LIN {X 0,Y 468.398,Z 466.939,A -85,B 0,C 180,E1 -7680.673,E2 -7680.673} C_VEL
LIN {X 0,Y 468.738,Z 461.358,A -85,B 0,C 180,E1 -7682.899,E2 -7682.899} C_VEL
LIN {X 0,Y 469.168,Z 453.805,A -85,B 0,C 180,E1 -7686.011,E2 -7686.011} C_VEL
LIN {X 0,Y 469.442,Z 448.312,A -85,B 0,C 180,E1 -7688.366,E2 -7688.366} C_VEL
LIN {X 0,Y 469.134,Z 444.309,A -85,B 0,C 180,E1 -7690.18,E2 -7690.18} C_VEL
LIN {X 0,Y 467.968,Z 437.991,A -85,B 0,C 180,E1 -7693.233,E2 -7693.233} C_VEL
LIN {X 0,Y 467.592,Z 435.867,A -85,B 0,C 180,E1 -7694.351,E2 -7694.351} C_VEL
LIN {X 0,Y 467.62,Z 435.861,A -85,B 0,C 180,E1 -7697.443,E2 -7697.443} C_VEL
LIN {X 0,Y 467.578,Z 435.869,A -85,B 0,C 180,E1 -7700.855,E2 -7700.855} C_VEL
LIN {X 0,Y 467.557,Z 435.868,A -85,B 0,C 180,E1 -7704.26,E2 -7704.26} C_VEL
LIN {X 0,Y 467.577,Z 435.869,A -85,B 0,C 180,E1 -7707.32,E2 -7707.32} C_VEL
LIN {X 0,Y 467.573,Z 435.868,A -85,B 0,C 180,E1 -7710.665,E2 -7710.665} C_VEL
LIN {X 0,Y 467.622,Z 435.862,A -85,B 0,C 180,E1 -7713.2,E2 -7713.2} C_VEL
LIN {X 0,Y 467.587,Z 435.866,A -85,B 0,C 180,E1 -7716.468,E2 -7716.468} C_VEL
LIN {X 0,Y 467.617,Z 435.862,A -85,B 0,C 180,E1 -7719.777,E2 -7719.777} C_VEL
LIN {X 0,Y 467.603,Z 435.866,A -85,B 0,C 180,E1 -7722.507,E2 -7722.507} C_VEL
LIN {X 0,Y 467.599,Z 435.866,A -85,B 0,C 180,E1 -7725.196,E2 -7725.196} C_VEL
LIN {X 0,Y 467.65,Z 435.858,A -85,B 0,C 180,E1 -7727.855,E2 -7727.855} C_VEL
LIN {X 0,Y 467.676,Z 435.854,A -85,B 0,C 180,E1 -7731.357,E2 -7731.357} C_VEL
LIN {X 0,Y 467.738,Z 435.847,A -85,B 0,C 180,E1 -7733.963,E2 -7733.963} C_VEL
LIN {X 0,Y 467.854,Z 435.833,A -85,B 0,C 180,E1 -7737.417,E2 -7737.417} C_VEL
LIN {X 0,Y 467.875,Z 435.829,A -85,B 0,C 180,E1 -7740,E2 -7740} C_VEL
LIN {X 0,Y 467.855,Z 435.833,A -85,B 0,C 180,E1 -7742.583,E2 -7742.583} C_VEL
LIN {X 0,Y 467.748,Z 435.848,A -85,B 0,C 180,E1 -7746.038,E2 -7746.038} C_VEL
LIN {X 0,Y 467.676,Z 435.857,A -85,B 0,C 180,E1 -7748.643,E2 -7748.643} C_VEL
LIN {X 0,Y 467.649,Z 435.858,A -85,B 0,C 180,E1 -7752.146,E2 -7752.146} C_VEL
LIN {X 0,Y 467.633,Z 435.861,A -85,B 0,C 180,E1 -7755.695,E2 -7755.695} C_VEL
LIN {X 0,Y 467.612,Z 435.863,A -85,B 0,C 180,E1 -7758.765,E2 -7758.765} C_VEL
LIN {X 0,Y 467.575,Z 435.867,A -85,B 0,C 180,E1 -7761.269,E2 -7761.269} C_VEL
LIN {X 0,Y 467.568,Z 435.871,A -85,B 0,C 180,E1 -7763.944,E2 -7763.944} C_VEL
LIN {X 0,Y 467.612,Z 435.862,A -85,B 0,C 180,E1 -7766.801,E2 -7766.801} C_VEL
LIN {X 0,Y 467.55,Z 435.871,A -85,B 0,C 180,E1 -7769.739,E2 -7769.739} C_VEL
LIN {X 0,Y 467.58,Z 435.867,A -85,B 0,C 180,E1 -7772.759,E2 -7772.759} C_VEL
LIN {X 0,Y 467.553,Z 435.871,A -85,B 0,C 180,E1 -7775.89,E2 -7775.89} C_VEL
LIN {X 0,Y 467.579,Z 435.867,A -85,B 0,C 180,E1 -7779.145,E2 -7779.145} C_VEL
LIN {X 0,Y 467.584,Z 435.867,A -85,B 0,C 180,E1 -7782.568,E2 -7782.568} C_VEL
LIN {X 0,Y 467.569,Z 435.866,A -85,B 0,C 180,E1 -7785.054,E2 -7785.054} C_VEL
LIN {X 0,Y 467.587,Z 435.867,A -85,B 0,C 180,E1 -7787.441,E2 -7787.441} C_VEL
LIN {X 0,Y 467.614,Z 435.862,A -85,B 0,C 180,E1 -7790.859,E2 -7790.859} C_VEL
LIN {X 0,Y 467.563,Z 435.869,A -85,B 0,C 180,E1 -7794.261,E2 -7794.261} C_VEL
LIN {X 0,Y 467.583,Z 435.866,A -85,B 0,C 180,E1 -7797.322,E2 -7797.322} C_VEL
LIN {X 0,Y 467.579,Z 435.867,A -85,B 0,C 180,E1 -7800.666,E2 -7800.666} C_VEL
LIN {X 0,Y 467.618,Z 435.861,A -85,B 0,C 180,E1 -7803.2,E2 -7803.2} C_VEL
LIN {X 0,Y 467.595,Z 435.865,A -85,B 0,C 180,E1 -7806.469,E2 -7806.469} C_VEL
LIN {X 0,Y 467.626,Z 435.862,A -85,B 0,C 180,E1 -7809.778,E2 -7809.778} C_VEL
LIN {X 0,Y 467.61,Z 435.861,A -85,B 0,C 180,E1 -7812.507,E2 -7812.507} C_VEL
LIN {X 0,Y 467.6,Z 435.863,A -85,B 0,C 180,E1 -7815.432,E2 -7815.432} C_VEL
LIN {X 0,Y 466.931,Z 435.948,A -85,B 0,C 180,E1 -7816.152,E2 -7816.152} C_VEL
LIN {X 0,Y 464.087,Z 436.304,A -85,B 0,C 180,E1 -7817.32,E2 -7817.32} C_VEL
LIN {X 0,Y 461.687,Z 436.602,A -85,B 0,C 180,E1 -7818.262,E2 -7818.262} C_VEL
LIN {X 0,Y 460.66,Z 436.73,A -85,B 0,C 180,E1 -7818.99,E2 -7818.99} C_VEL
LIN {X 0,Y 460.578,Z 436.738,A -85,B 0,C 180,E1 -7819.236,E2 -7819.236} C_VEL
LIN {X 0,Y 460.673,Z 436.727,A -85,B 0,C 180,E1 -7822.588,E2 -7822.588} C_VEL
LIN {X 0,Y 460.694,Z 436.724,A -85,B 0,C 180,E1 -7824.748,E2 -7824.748} C_VEL
LIN {X 0,Y 460.828,Z 436.709,A -85,B 0,C 180,E1 -7827.378,E2 -7827.378} C_VEL
LIN {X 0,Y 460.857,Z 436.703,A -85,B 0,C 180,E1 -7830,E2 -7830} C_VEL
LIN {X 0,Y 460.804,Z 436.711,A -85,B 0,C 180,E1 -7832.622,E2 -7832.622} C_VEL
LIN {X 0,Y 460.712,Z 436.722,A -85,B 0,C 180,E1 -7836.13,E2 -7836.13} C_VEL
LIN {X 0,Y 460.625,Z 436.733,A -85,B 0,C 180,E1 -7838.776,E2 -7838.776} C_VEL
LIN {X 0,Y 460.617,Z 436.734,A -85,B 0,C 180,E1 -7842.445,E2 -7842.445} C_VEL
LIN {X 0,Y 460.603,Z 436.736,A -85,B 0,C 180,E1 -7845.997,E2 -7845.997} C_VEL
LIN {X 0,Y 460.574,Z 436.741,A -85,B 0,C 180,E1 -7848.901,E2 -7848.901} C_VEL
LIN {X 0,Y 460.518,Z 436.749,A -85,B 0,C 180,E1 -7851.485,E2 -7851.485} C_VEL
LIN {X 0,Y 460.545,Z 436.743,A -85,B 0,C 180,E1 -7854.332,E2 -7854.332} C_VEL
LIN {X 0,Y 460.581,Z 436.74,A -85,B 0,C 180,E1 -7857.243,E2 -7857.243} C_VEL
LIN {X 0,Y 460.512,Z 436.748,A -85,B 0,C 180,E1 -7860.239,E2 -7860.239} C_VEL
LIN {X 0,Y 460.505,Z 436.748,A -85,B 0,C 180,E1 -7863.326,E2 -7863.326} C_VEL
LIN {X 0,Y 460.311,Z 436.774,A -85,B 0,C 180,E1 -7865.981,E2 -7865.981} C_VEL
LIN {X 0,Y 459.97,Z 436.818,A -85,B 0,C 180,E1 -7868.808,E2 -7868.808} C_VEL
LIN {X 0,Y 459.875,Z 438.549,A -85,B 0,C 180,E1 -7871.081,E2 -7871.081} C_VEL
LIN {X 0,Y 459.846,Z 441.335,A -85,B 0,C 180,E1 -7874.084,E2 -7874.084} C_VEL
LIN {X 0,Y 459.801,Z 444.258,A -85,B 0,C 180,E1 -7877.194,E2 -7877.194} C_VEL
LIN {X 0,Y 459.741,Z 446.977,A -85,B 0,C 180,E1 -7880.055,E2 -7880.055} C_VEL
LIN {X 0,Y 459.739,Z 450.158,A -85,B 0,C 180,E1 -7883.225,E2 -7883.225} C_VEL
LIN {X 0,Y 463.705,Z 464.798,A -85,B 0,C 180,E1 -7883.796,E2 -7883.796} C_VEL
LIN {X 0,Y 464.998,Z 471.275,A -85,B 0,C 180,E1 -7884.091,E2 -7884.091} C_VEL
LIN {X 0,Y 464.463,Z 485.389,A -85,B 0,C 180,E1 -7884.736,E2 -7884.736} C_VEL
LIN {X 0,Y 463.818,Z 498.227,A -85,B 0,C 180,E1 -7885.505,E2 -7885.505} C_VEL
LIN {X 0,Y 463.147,Z 510.816,A -85,B 0,C 180,E1 -7886.457,E2 -7886.457} C_VEL
LIN {X 0,Y 462.369,Z 523.07,A -85,B 0,C 180,E1 -7887.602,E2 -7887.602} C_VEL
LIN {X 0,Y 461.745,Z 533.858,A -85,B 0,C 180,E1 -7888.835,E2 -7888.835} C_VEL
LIN {X 0,Y 461.179,Z 543.327,A -85,B 0,C 180,E1 -7890.144,E2 -7890.144} C_VEL
LIN {X 0,Y 460.683,Z 551.611,A -85,B 0,C 180,E1 -7891.527,E2 -7891.527} C_VEL
LIN {X 0,Y 460.316,Z 558.783,A -85,B 0,C 180,E1 -7892.985,E2 -7892.985} C_VEL
LIN {X 0,Y 460.008,Z 565.432,A -85,B 0,C 180,E1 -7894.673,E2 -7894.673} C_VEL
LIN {X 0,Y 459.828,Z 569.82,A -85,B 0,C 180,E1 -7896.107,E2 -7896.107} C_VEL
LIN {X 0,Y 459.652,Z 573.148,A -85,B 0,C 180,E1 -7897.527,E2 -7897.527} C_VEL
LIN {X 0,Y 459.541,Z 576.153,A -85,B 0,C 180,E1 -7899.405,E2 -7899.405} C_VEL
LIN {X 0,Y 459.512,Z 577.582,A -85,B 0,C 180,E1 -7901.265,E2 -7901.265} C_VEL
LIN {X 0,Y 459.48,Z 577.505,A -85,B 0,C 180,E1 -7903.105,E2 -7903.105} C_VEL
LIN {X 0,Y 459.542,Z 575.992,A -85,B 0,C 180,E1 -7904.93,E2 -7904.93} C_VEL
LIN {X 0,Y 459.658,Z 573.047,A -85,B 0,C 180,E1 -7906.741,E2 -7906.741} C_VEL
LIN {X 0,Y 459.847,Z 570.13,A -85,B 0,C 180,E1 -7907.991,E2 -7907.991} C_VEL
LIN {X 0,Y 460.019,Z 565.795,A -85,B 0,C 180,E1 -7909.436,E2 -7909.436} C_VEL
LIN {X 0,Y 460.316,Z 560.71,A -85,B 0,C 180,E1 -7910.775,E2 -7910.775} C_VEL
LIN {X 0,Y 460.662,Z 553.602,A -85,B 0,C 180,E1 -7912.304,E2 -7912.304} C_VEL
LIN {X 0,Y 461.186,Z 545.878,A -85,B 0,C 180,E1 -7913.657,E2 -7913.657} C_VEL
LIN {X 0,Y 461.679,Z 536.828,A -85,B 0,C 180,E1 -7914.978,E2 -7914.978} C_VEL
LIN {X 0,Y 462.26,Z 527.811,A -85,B 0,C 180,E1 -7916.077,E2 -7916.077} C_VEL
LIN {X 0,Y 462.946,Z 517.097,A -85,B 0,C 180,E1 -7917.172,E2 -7917.172} C_VEL
LIN {X 0,Y 463.623,Z 505.448,A -85,B 0,C 180,E1 -7918.154,E2 -7918.154} C_VEL
LIN {X 0,Y 464.273,Z 493.279,A -85,B 0,C 180,E1 -7918.985,E2 -7918.985} C_VEL
LIN {X 0,Y 464.898,Z 479.944,A -85,B 0,C 180,E1 -7919.701,E2 -7919.701} C_VEL
LIN {X 0,Y 465.049,Z 470.104,A -85,B 0,C 180,E1 -7920.122,E2 -7920.122} C_VEL
LIN {X 0,Y 461.6,Z 457.575,A -85,B 0,C 180,E1 -7920.692,E2 -7920.692} C_VEL
LIN {X 0,Y 459.896,Z 451.959,A -85,B 0,C 180,E1 -7920.93,E2 -7920.93} C_VEL
LIN {X 0,Y 460.184,Z 449.053,A -85,B 0,C 180,E1 -7924.379,E2 -7924.379} C_VEL
LIN {X 0,Y 460.258,Z 446.91,A -85,B 0,C 180,E1 -7927.016,E2 -7927.016} C_VEL
LIN {X 0,Y 460.23,Z 444.85,A -85,B 0,C 180,E1 -7929.67,E2 -7929.67} C_VEL
LIN {X 0,Y 460.37,Z 442.807,A -85,B 0,C 180,E1 -7932.341,E2 -7932.341} C_VEL
LIN {X 0,Y 460.427,Z 440.21,A -85,B 0,C 180,E1 -7935.947,E2 -7935.947} C_VEL
LIN {X 0,Y 460.603,Z 438.172,A -85,B 0,C 180,E1 -7938.916,E2 -7938.916} C_VEL
LIN {X 0,Y 460.5,Z 436.752,A -85,B 0,C 180,E1 -7941.486,E2 -7941.486} C_VEL
LIN {X 0,Y 460.537,Z 436.747,A -85,B 0,C 180,E1 -7944.332,E2 -7944.332} C_VEL
LIN {X 0,Y 460.578,Z 436.74,A -85,B 0,C 180,E1 -7947.243,E2 -7947.243} C_VEL
LIN {X 0,Y 460.522,Z 436.748,A -85,B 0,C 180,E1 -7950.239,E2 -7950.239} C_VEL
LIN {X 0,Y 460.524,Z 436.746,A -85,B 0,C 180,E1 -7953.325,E2 -7953.325} C_VEL
LIN {X 0,Y 460.474,Z 436.753,A -85,B 0,C 180,E1 -7956.53,E2 -7956.53} C_VEL
LIN {X 0,Y 460.572,Z 436.743,A -85,B 0,C 180,E1 -7959.858,E2 -7959.858} C_VEL
LIN {X 0,Y 460.544,Z 436.746,A -85,B 0,C 180,E1 -7962.179,E2 -7962.179} C_VEL
LIN {X 0,Y 460.701,Z 437.663,A -85,B 0,C 180,E1 -7963.352,E2 -7963.352} C_VEL
LIN {X 0,Y 461.163,Z 440.423,A -85,B 0,C 180,E1 -7965.747,E2 -7965.747} C_VEL
LIN {X 0,Y 461.796,Z 443.856,A -85,B 0,C 180,E1 -7968.221,E2 -7968.221} C_VEL
LIN {X 0,Y 462.269,Z 447.226,A -85,B 0,C 180,E1 -7970.318,E2 -7970.318} C_VEL
LIN {X 0,Y 462.362,Z 450.715,A -85,B 0,C 180,E1 -7972.224,E2 -7972.224} C_VEL
LIN {X 0,Y 461.729,Z 457.028,A -85,B 0,C 180,E1 -7975.279,E2 -7975.279} C_VEL
LIN {X 0,Y 461.397,Z 462.642,A -85,B 0,C 180,E1 -7977.784,E2 -7977.784} C_VEL
LIN {X 0,Y 460.967,Z 469.887,A -85,B 0,C 180,E1 -7980.799,E2 -7980.799} C_VEL
LIN {X 0,Y 460.603,Z 478.552,A -85,B 0,C 180,E1 -7984.189,E2 -7984.189} C_VEL
LIN {X 0,Y 460.323,Z 487.611,A -85,B 0,C 180,E1 -7987.562,E2 -7987.562} C_VEL
LIN {X 0,Y 460.101,Z 497.269,A -85,B 0,C 180,E1 -7991.036,E2 -7991.036} C_VEL
LIN {X 0,Y 463.252,Z 515.79,A -85,B 0,C 180,E1 -7991.68,E2 -7991.68} C_VEL
LIN {X 0,Y 464.612,Z 524.172,A -85,B 0,C 180,E1 -7992.049,E2 -7992.049} C_VEL
LIN {X 0,Y 463.983,Z 537.899,A -85,B 0,C 180,E1 -7992.69,E2 -7992.69} C_VEL
LIN {X 0,Y 463.294,Z 550.907,A -85,B 0,C 180,E1 -7993.476,E2 -7993.476} C_VEL
LIN {X 0,Y 462.523,Z 563.982,A -85,B 0,C 180,E1 -7994.466,E2 -7994.466} C_VEL
LIN {X 0,Y 461.782,Z 575.862,A -85,B 0,C 180,E1 -7995.569,E2 -7995.569} C_VEL
LIN {X 0,Y 461.204,Z 586.667,A -85,B 0,C 180,E1 -7996.787,E2 -7996.787} C_VEL
LIN {X 0,Y 460.751,Z 596.45,A -85,B 0,C 180,E1 -7998.117,E2 -7998.117} C_VEL
LIN {X 0,Y 460.226,Z 605.805,A -85,B 0,C 180,E1 -7999.664,E2 -7999.664} C_VEL
LIN {X 0,Y 459.939,Z 613.344,A -85,B 0,C 180,E1 -8001.211,E2 -8001.211} C_VEL
LIN {X 0,Y 459.733,Z 620.127,A -85,B 0,C 180,E1 -8002.975,E2 -8002.975} C_VEL
LIN {X 0,Y 459.694,Z 625.223,A -85,B 0,C 180,E1 -8004.737,E2 -8004.737} C_VEL
LIN {X 0,Y 459.645,Z 628.777,A -85,B 0,C 180,E1 -8006.494,E2 -8006.494} C_VEL
LIN {X 0,Y 459.624,Z 630.897,A -85,B 0,C 180,E1 -8008.248,E2 -8008.248} C_VEL
LIN {X 0,Y 459.528,Z 631.621,A -85,B 0,C 180,E1 -8010,E2 -8010} C_VEL
LIN {X 0,Y 459.624,Z 630.975,A -85,B 0,C 180,E1 -8011.752,E2 -8011.752} C_VEL
LIN {X 0,Y 459.613,Z 628.939,A -85,B 0,C 180,E1 -8013.507,E2 -8013.507} C_VEL
LIN {X 0,Y 459.672,Z 625.476,A -85,B 0,C 180,E1 -8015.263,E2 -8015.263} C_VEL
LIN {X 0,Y 459.731,Z 620.478,A -85,B 0,C 180,E1 -8017.025,E2 -8017.025} C_VEL
LIN {X 0,Y 459.939,Z 613.811,A -85,B 0,C 180,E1 -8018.789,E2 -8018.789} C_VEL
LIN {X 0,Y 460.236,Z 606.382,A -85,B 0,C 180,E1 -8020.336,E2 -8020.336} C_VEL
LIN {X 0,Y 460.746,Z 597.146,A -85,B 0,C 180,E1 -8021.883,E2 -8021.883} C_VEL
LIN {X 0,Y 461.219,Z 587.487,A -85,B 0,C 180,E1 -8023.213,E2 -8023.213} C_VEL
LIN {X 0,Y 461.897,Z 576.811,A -85,B 0,C 180,E1 -8024.427,E2 -8024.427} C_VEL
LIN {X 0,Y 462.614,Z 565.044,A -85,B 0,C 180,E1 -8025.531,E2 -8025.531} C_VEL
LIN {X 0,Y 463.39,Z 552.023,A -85,B 0,C 180,E1 -8026.521,E2 -8026.521} C_VEL
LIN {X 0,Y 464.056,Z 539.426,A -85,B 0,C 180,E1 -8027.283,E2 -8027.283} C_VEL
LIN {X 0,Y 464.621,Z 525.111,A -85,B 0,C 180,E1 -8027.95,E2 -8027.95} C_VEL
LIN {X 0,Y 462.452,Z 511.225,A -85,B 0,C 180,E1 -8028.512,E2 -8028.512} C_VEL
LIN {X 0,Y 460.134,Z 499.005,A -85,B 0,C 180,E1 -8028.892,E2 -8028.892} C_VEL
LIN {X 0,Y 460.377,Z 490.633,A -85,B 0,C 180,E1 -8031.963,E2 -8031.963} C_VEL
LIN {X 0,Y 460.741,Z 481.777,A -85,B 0,C 180,E1 -8035.283,E2 -8035.283} C_VEL
LIN {X 0,Y 461.037,Z 474.214,A -85,B 0,C 180,E1 -8038.2,E2 -8038.2} C_VEL
LIN {X 0,Y 461.541,Z 465.915,A -85,B 0,C 180,E1 -8041.491,E2 -8041.491} C_VEL
LIN {X 0,Y 461.932,Z 457.996,A -85,B 0,C 180,E1 -8044.757,E2 -8044.757} C_VEL
LIN {X 0,Y 462.425,Z 450.94,A -85,B 0,C 180,E1 -8047.786,E2 -8047.786} C_VEL
LIN {X 0,Y 462.324,Z 446.742,A -85,B 0,C 180,E1 -8049.676,E2 -8049.676} C_VEL
LIN {X 0,Y 461.467,Z 441.777,A -85,B 0,C 180,E1 -8052.074,E2 -8052.074} C_VEL
LIN {X 0,Y 460.54,Z 436.746,A -85,B 0,C 180,E1 -8054.657,E2 -8054.657} C_VEL
LIN {X 0,Y 460.543,Z 436.743,A -85,B 0,C 180,E1 -8057.821,E2 -8057.821} C_VEL
LIN {X 0,Y 460.54,Z 436.744,A -85,B 0,C 180,E1 -8061.102,E2 -8061.102} C_VEL
LIN {X 0,Y 460.508,Z 436.748,A -85,B 0,C 180,E1 -8064.554,E2 -8064.554} C_VEL
LIN {X 0,Y 460.528,Z 436.744,A -85,B 0,C 180,E1 -8067.715,E2 -8067.715} C_VEL
LIN {X 0,Y 460.542,Z 436.744,A -85,B 0,C 180,E1 -8070.769,E2 -8070.769} C_VEL
LIN {X 0,Y 460.562,Z 436.741,A -85,B 0,C 180,E1 -8073.735,E2 -8073.735} C_VEL
LIN {X 0,Y 460.54,Z 436.744,A -85,B 0,C 180,E1 -8076.624,E2 -8076.624} C_VEL
LIN {X 0,Y 460.546,Z 436.745,A -85,B 0,C 180,E1 -8079.453,E2 -8079.453} C_VEL
LIN {X 0,Y 460.553,Z 436.741,A -85,B 0,C 180,E1 -8082.23,E2 -8082.23} C_VEL
LIN {X 0,Y 460.558,Z 436.743,A -85,B 0,C 180,E1 -8084.965,E2 -8084.965} C_VEL
LIN {X 0,Y 460.607,Z 436.736,A -85,B 0,C 180,E1 -8088.559,E2 -8088.559} C_VEL
LIN {X 0,Y 460.688,Z 436.726,A -85,B 0,C 180,E1 -8092.109,E2 -8092.109} C_VEL
LIN {X 0,Y 460.692,Z 436.727,A -85,B 0,C 180,E1 -8094.748,E2 -8094.748} C_VEL
LIN {X 0,Y 460.819,Z 436.71,A -85,B 0,C 180,E1 -8097.378,E2 -8097.378} C_VEL
LIN {X 0,Y 460.846,Z 436.704,A -85,B 0,C 180,E1 -8100,E2 -8100} C_VEL
LIN {X 0,Y 460.82,Z 436.71,A -85,B 0,C 180,E1 -8102.623,E2 -8102.623} C_VEL
LIN {X 0,Y 460.712,Z 436.724,A -85,B 0,C 180,E1 -8106.13,E2 -8106.13} C_VEL
LIN {X 0,Y 460.623,Z 436.734,A -85,B 0,C 180,E1 -8108.776,E2 -8108.776} C_VEL
LIN {X 0,Y 460.607,Z 436.737,A -85,B 0,C 180,E1 -8112.445,E2 -8112.445} C_VEL
LIN {X 0,Y 460.594,Z 436.738,A -85,B 0,C 180,E1 -8115.998,E2 -8115.998} C_VEL
LIN {X 0,Y 460.565,Z 436.74,A -85,B 0,C 180,E1 -8118.902,E2 -8118.902} C_VEL
LIN {X 0,Y 460.511,Z 436.747,A -85,B 0,C 180,E1 -8121.486,E2 -8121.486} C_VEL
LIN {X 0,Y 460.538,Z 436.745,A -85,B 0,C 180,E1 -8124.333,E2 -8124.333} C_VEL
LIN {X 0,Y 460.568,Z 436.738,A -85,B 0,C 180,E1 -8127.244,E2 -8127.244} C_VEL
LIN {X 0,Y 460.507,Z 436.749,A -85,B 0,C 180,E1 -8130.241,E2 -8130.241} C_VEL
LIN {X 0,Y 460.526,Z 436.746,A -85,B 0,C 180,E1 -8133.325,E2 -8133.325} C_VEL
LIN {X 0,Y 460.475,Z 436.752,A -85,B 0,C 180,E1 -8136.53,E2 -8136.53} C_VEL
LIN {X 0,Y 460.542,Z 436.744,A -85,B 0,C 180,E1 -8138.898,E2 -8138.898} C_VEL
LIN {X 0,Y 460.521,Z 436.747,A -85,B 0,C 180,E1 -8142.182,E2 -8142.182} C_VEL
LIN {X 0,Y 460.515,Z 436.746,A -85,B 0,C 180,E1 -8145.412,E2 -8145.412} C_VEL
LIN {X 0,Y 460.534,Z 436.746,A -85,B 0,C 180,E1 -8148.398,E2 -8148.398} C_VEL
LIN {X 0,Y 460.543,Z 436.744,A -85,B 0,C 180,E1 -8151.269,E2 -8151.269} C_VEL
LIN {X 0,Y 460.514,Z 436.746,A -85,B 0,C 180,E1 -8154.555,E2 -8154.555} C_VEL
LIN {X 0,Y 460.533,Z 436.746,A -85,B 0,C 180,E1 -8157.716,E2 -8157.716} C_VEL
LIN {X 0,Y 460.548,Z 436.743,A -85,B 0,C 180,E1 -8160.77,E2 -8160.77} C_VEL
LIN {X 0,Y 460.565,Z 436.743,A -85,B 0,C 180,E1 -8163.735,E2 -8163.735} C_VEL
LIN {X 0,Y 460.548,Z 436.742,A -85,B 0,C 180,E1 -8166.625,E2 -8166.625} C_VEL
LIN {X 0,Y 460.554,Z 436.743,A -85,B 0,C 180,E1 -8169.453,E2 -8169.453} C_VEL
LIN {X 0,Y 460.561,Z 436.74,A -85,B 0,C 180,E1 -8172.231,E2 -8172.231} C_VEL
LIN {X 0,Y 460.569,Z 436.741,A -85,B 0,C 180,E1 -8174.965,E2 -8174.965} C_VEL
LIN {X 0,Y 460.614,Z 436.734,A -85,B 0,C 180,E1 -8178.56,E2 -8178.56} C_VEL
LIN {X 0,Y 460.578,Z 436.738,A -85,B 0,C 180,E1 -8179.236,E2 -8179.236} C_VEL
LIN {X 0,Y 459.916,Z 436.824,A -85,B 0,C 180,E1 -8179.966,E2 -8179.966} C_VEL
LIN {X 0,Y 457.075,Z 437.179,A -85,B 0,C 180,E1 -8181.152,E2 -8181.152} C_VEL
LIN {X 0,Y 454.682,Z 437.476,A -85,B 0,C 180,E1 -8182.109,E2 -8182.109} C_VEL
LIN {X 0,Y 453.672,Z 437.6,A -85,B 0,C 180,E1 -8182.848,E2 -8182.848} C_VEL
LIN {X 0,Y 453.599,Z 437.608,A -85,B 0,C 180,E1 -8183.098,E2 -8183.098} C_VEL
LIN {X 0,Y 453.666,Z 437.6,A -85,B 0,C 180,E1 -8184.667,E2 -8184.667} C_VEL
LIN {X 0,Y 453.769,Z 437.588,A -85,B 0,C 180,E1 -8187.337,E2 -8187.337} C_VEL
LIN {X 0,Y 453.827,Z 437.579,A -85,B 0,C 180,E1 -8190,E2 -8190} C_VEL
LIN {X 0,Y 453.748,Z 437.59,A -85,B 0,C 180,E1 -8192.663,E2 -8192.663} C_VEL
LIN {X 0,Y 453.678,Z 437.598,A -85,B 0,C 180,E1 -8196.225,E2 -8196.225} C_VEL
LIN {X 0,Y 453.59,Z 437.609,A -85,B 0,C 180,E1 -8198.913,E2 -8198.913} C_VEL
LIN {X 0,Y 453.567,Z 437.613,A -85,B 0,C 180,E1 -8202.529,E2 -8202.529} C_VEL
LIN {X 0,Y 453.548,Z 437.615,A -85,B 0,C 180,E1 -8206.196,E2 -8206.196} C_VEL
LIN {X 0,Y 453.523,Z 437.62,A -85,B 0,C 180,E1 -8209.04,E2 -8209.04} C_VEL
LIN {X 0,Y 453.479,Z 437.623,A -85,B 0,C 180,E1 -8211.836,E2 -8211.836} C_VEL
LIN {X 0,Y 453.516,Z 437.62,A -85,B 0,C 180,E1 -8214.734,E2 -8214.734} C_VEL
LIN {X 0,Y 453.539,Z 437.614,A -85,B 0,C 180,E1 -8217.96,E2 -8217.96} C_VEL
LIN {X 0,Y 453.464,Z 437.624,A -85,B 0,C 180,E1 -8221.524,E2 -8221.524} C_VEL
LIN {X 0,Y 453.437,Z 437.628,A -85,B 0,C 180,E1 -8223.915,E2 -8223.915} C_VEL
LIN {X 0,Y 453.239,Z 437.655,A -85,B 0,C 180,E1 -8226.261,E2 -8226.261} C_VEL
LIN {X 0,Y 452.827,Z 437.821,A -85,B 0,C 180,E1 -8229.518,E2 -8229.518} C_VEL
LIN {X 0,Y 452.81,Z 441.061,A -85,B 0,C 180,E1 -8233.071,E2 -8233.071} C_VEL
LIN {X 0,Y 452.739,Z 443.499,A -85,B 0,C 180,E1 -8235.689,E2 -8235.689} C_VEL
LIN {X 0,Y 452.698,Z 445.841,A -85,B 0,C 180,E1 -8238.174,E2 -8238.174} C_VEL
LIN {X 0,Y 452.619,Z 449.099,A -85,B 0,C 180,E1 -8241.603,E2 -8241.603} C_VEL
LIN {X 0,Y 452.631,Z 450.374,A -85,B 0,C 180,E1 -8242.912,E2 -8242.912} C_VEL
LIN {X 0,Y 457.129,Z 466.893,A -85,B 0,C 180,E1 -8243.596,E2 -8243.596} C_VEL
LIN {X 0,Y 458.231,Z 471.932,A -85,B 0,C 180,E1 -8243.842,E2 -8243.842} C_VEL
LIN {X 0,Y 457.666,Z 486.107,A -85,B 0,C 180,E1 -8244.506,E2 -8244.506} C_VEL
LIN {X 0,Y 456.96,Z 499.267,A -85,B 0,C 180,E1 -8245.315,E2 -8245.315} C_VEL
LIN {X 0,Y 456.219,Z 512.158,A -85,B 0,C 180,E1 -8246.318,E2 -8246.318} C_VEL
LIN {X 0,Y 455.449,Z 523.903,A -85,B 0,C 180,E1 -8247.444,E2 -8247.444} C_VEL
LIN {X 0,Y 454.864,Z 533.613,A -85,B 0,C 180,E1 -8248.569,E2 -8248.569} C_VEL
LIN {X 0,Y 454.225,Z 543.645,A -85,B 0,C 180,E1 -8249.967,E2 -8249.967} C_VEL
LIN {X 0,Y 453.686,Z 551.566,A -85,B 0,C 180,E1 -8251.3,E2 -8251.3} C_VEL
LIN {X 0,Y 453.319,Z 558.831,A -85,B 0,C 180,E1 -8252.783,E2 -8252.783} C_VEL
LIN {X 0,Y 452.979,Z 564.681,A -85,B 0,C 180,E1 -8254.251,E2 -8254.251} C_VEL
LIN {X 0,Y 452.796,Z 569.335,A -85,B 0,C 180,E1 -8255.712,E2 -8255.712} C_VEL
LIN {X 0,Y 452.613,Z 572.925,A -85,B 0,C 180,E1 -8257.158,E2 -8257.158} C_VEL
LIN {X 0,Y 452.473,Z 576.169,A -85,B 0,C 180,E1 -8259.069,E2 -8259.069} C_VEL
LIN {X 0,Y 452.423,Z 577.852,A -85,B 0,C 180,E1 -8260.96,E2 -8260.96} C_VEL
LIN {X 0,Y 452.396,Z 578.052,A -85,B 0,C 180,E1 -8262.832,E2 -8262.832} C_VEL
LIN {X 0,Y 452.461,Z 576.772,A -85,B 0,C 180,E1 -8264.689,E2 -8264.689} C_VEL
LIN {X 0,Y 452.574,Z 574.036,A -85,B 0,C 180,E1 -8266.53,E2 -8266.53} C_VEL
LIN {X 0,Y 452.774,Z 570.99,A -85,B 0,C 180,E1 -8267.925,E2 -8267.925} C_VEL
LIN {X 0,Y 453.005,Z 565.622,A -85,B 0,C 180,E1 -8269.722,E2 -8269.722} C_VEL
LIN {X 0,Y 453.339,Z 560.458,A -85,B 0,C 180,E1 -8271.081,E2 -8271.081} C_VEL
LIN {X 0,Y 453.772,Z 552.92,A -85,B 0,C 180,E1 -8272.681,E2 -8272.681} C_VEL
LIN {X 0,Y 454.288,Z 545.31,A -85,B 0,C 180,E1 -8274.006,E2 -8274.006} C_VEL
LIN {X 0,Y 454.892,Z 536.025,A -85,B 0,C 180,E1 -8275.347,E2 -8275.347} C_VEL
LIN {X 0,Y 455.604,Z 525.772,A -85,B 0,C 180,E1 -8276.573,E2 -8276.573} C_VEL
LIN {X 0,Y 456.313,Z 514.54,A -85,B 0,C 180,E1 -8277.683,E2 -8277.683} C_VEL
LIN {X 0,Y 457.072,Z 501.895,A -85,B 0,C 180,E1 -8278.7,E2 -8278.7} C_VEL
LIN {X 0,Y 457.75,Z 488.595,A -85,B 0,C 180,E1 -8279.552,E2 -8279.552} C_VEL
LIN {X 0,Y 458.416,Z 474.517,A -85,B 0,C 180,E1 -8280.241,E2 -8280.241} C_VEL
LIN {X 0,Y 458.227,Z 470.76,A -85,B 0,C 180,E1 -8280.405,E2 -8280.405} C_VEL
LIN {X 0,Y 454.439,Z 457.521,A -85,B 0,C 180,E1 -8281.038,E2 -8281.038} C_VEL
LIN {X 0,Y 452.821,Z 452.507,A -85,B 0,C 180,E1 -8281.25,E2 -8281.25} C_VEL
LIN {X 0,Y 453.148,Z 449.854,A -85,B 0,C 180,E1 -8284.447,E2 -8284.447} C_VEL
LIN {X 0,Y 453.214,Z 447.722,A -85,B 0,C 180,E1 -8287.126,E2 -8287.126} C_VEL
LIN {X 0,Y 453.186,Z 445.66,A -85,B 0,C 180,E1 -8289.822,E2 -8289.822} C_VEL
LIN {X 0,Y 453.32,Z 443.64,A -85,B 0,C 180,E1 -8292.536,E2 -8292.536} C_VEL
LIN {X 0,Y 453.412,Z 441.053,A -85,B 0,C 180,E1 -8296.201,E2 -8296.201} C_VEL
LIN {X 0,Y 453.593,Z 439.161,A -85,B 0,C 180,E1 -8299.07,E2 -8299.07} C_VEL
LIN {X 0,Y 453.465,Z 437.628,A -85,B 0,C 180,E1 -8301.837,E2 -8301.837} C_VEL
LIN {X 0,Y 453.508,Z 437.621,A -85,B 0,C 180,E1 -8304.735,E2 -8304.735} C_VEL
LIN {X 0,Y 453.533,Z 437.619,A -85,B 0,C 180,E1 -8307.962,E2 -8307.962} C_VEL
LIN {X 0,Y 453.478,Z 437.624,A -85,B 0,C 180,E1 -8310.759,E2 -8310.759} C_VEL
LIN {X 0,Y 453.473,Z 437.625,A -85,B 0,C 180,E1 -8313.913,E2 -8313.913} C_VEL
LIN {X 0,Y 453.466,Z 437.626,A -85,B 0,C 180,E1 -8317.188,E2 -8317.188} C_VEL
LIN {X 0,Y 453.527,Z 437.619,A -85,B 0,C 180,E1 -8319.446,E2 -8319.446} C_VEL
LIN {X 0,Y 453.54,Z 437.897,A -85,B 0,C 180,E1 -8321.945,E2 -8321.945} C_VEL
LIN {X 0,Y 454.016,Z 440.58,A -85,B 0,C 180,E1 -8324.598,E2 -8324.598} C_VEL
LIN {X 0,Y 454.743,Z 444.815,A -85,B 0,C 180,E1 -8327.888,E2 -8327.888} C_VEL
LIN {X 0,Y 455.213,Z 447.406,A -85,B 0,C 180,E1 -8329.577,E2 -8329.577} C_VEL
LIN {X 0,Y 455.415,Z 450.379,A -85,B 0,C 180,E1 -8331.319,E2 -8331.319} C_VEL
LIN {X 0,Y 455.088,Z 454.38,A -85,B 0,C 180,E1 -8333.422,E2 -8333.422} C_VEL
LIN {X 0,Y 454.527,Z 461.11,A -85,B 0,C 180,E1 -8336.612,E2 -8336.612} C_VEL
LIN {X 0,Y 454.112,Z 467.219,A -85,B 0,C 180,E1 -8339.289,E2 -8339.289} C_VEL
LIN {X 0,Y 453.747,Z 474.573,A -85,B 0,C 180,E1 -8342.312,E2 -8342.312} C_VEL
LIN {X 0,Y 453.429,Z 482.105,A -85,B 0,C 180,E1 -8345.261,E2 -8345.261} C_VEL
LIN {X 0,Y 453.169,Z 490.763,A -85,B 0,C 180,E1 -8348.515,E2 -8348.515} C_VEL
LIN {X 0,Y 453.024,Z 496.747,A -85,B 0,C 180,E1 -8350.702,E2 -8350.702} C_VEL
LIN {X 0,Y 456.101,Z 514.227,A -85,B 0,C 180,E1 -8351.338,E2 -8351.338} C_VEL
LIN {X 0,Y 457.77,Z 525.816,A -85,B 0,C 180,E1 -8351.86,E2 -8351.86} C_VEL
LIN {X 0,Y 457.098,Z 538.869,A -85,B 0,C 180,E1 -8352.501,E2 -8352.501} C_VEL
LIN {X 0,Y 456.358,Z 552.055,A -85,B 0,C 180,E1 -8353.332,E2 -8353.332} C_VEL
LIN {X 0,Y 455.539,Z 564.834,A -85,B 0,C 180,E1 -8354.337,E2 -8354.337} C_VEL
LIN {X 0,Y 454.766,Z 576.461,A -85,B 0,C 180,E1 -8355.456,E2 -8355.456} C_VEL
LIN {X 0,Y 454.22,Z 586.157,A -85,B 0,C 180,E1 -8356.58,E2 -8356.58} C_VEL
LIN {X 0,Y 453.755,Z 595.936,A -85,B 0,C 180,E1 -8357.931,E2 -8357.931} C_VEL
LIN {X 0,Y 453.191,Z 605.313,A -85,B 0,C 180,E1 -8359.501,E2 -8359.501} C_VEL
LIN {X 0,Y 452.891,Z 612.871,A -85,B 0,C 180,E1 -8361.073,E2 -8361.073} C_VEL
LIN {X 0,Y 452.651,Z 619.671,A -85,B 0,C 180,E1 -8362.865,E2 -8362.865} C_VEL
LIN {X 0,Y 452.6,Z 624.782,A -85,B 0,C 180,E1 -8364.654,E2 -8364.654} C_VEL
LIN {X 0,Y 452.542,Z 628.348,A -85,B 0,C 180,E1 -8366.439,E2 -8366.439} C_VEL
LIN {X 0,Y 452.532,Z 630.478,A -85,B 0,C 180,E1 -8368.22,E2 -8368.22} C_VEL
LIN {X 0,Y 452.462,Z 631.206,A -85,B 0,C 180,E1 -8370,E2 -8370} C_VEL
LIN {X 0,Y 452.532,Z 630.559,A -85,B 0,C 180,E1 -8371.78,E2 -8371.78} C_VEL
LIN {X 0,Y 452.513,Z 628.519,A -85,B 0,C 180,E1 -8373.562,E2 -8373.562} C_VEL
LIN {X 0,Y 452.583,Z 625.049,A -85,B 0,C 180,E1 -8375.346,E2 -8375.346} C_VEL
LIN {X 0,Y 452.651,Z 620.04,A -85,B 0,C 180,E1 -8377.135,E2 -8377.135} C_VEL
LIN {X 0,Y 452.885,Z 613.358,A -85,B 0,C 180,E1 -8378.927,E2 -8378.927} C_VEL
LIN {X 0,Y 453.207,Z 605.913,A -85,B 0,C 180,E1 -8380.498,E2 -8380.498} C_VEL
LIN {X 0,Y 453.754,Z 596.653,A -85,B 0,C 180,E1 -8382.069,E2 -8382.069} C_VEL
LIN {X 0,Y 454.234,Z 586.972,A -85,B 0,C 180,E1 -8383.419,E2 -8383.419} C_VEL
LIN {X 0,Y 454.912,Z 576.271,A -85,B 0,C 180,E1 -8384.654,E2 -8384.654} C_VEL
LIN {X 0,Y 455.693,Z 564.485,A -85,B 0,C 180,E1 -8385.773,E2 -8385.773} C_VEL
LIN {X 0,Y 456.537,Z 551.444,A -85,B 0,C 180,E1 -8386.776,E2 -8386.776} C_VEL
LIN {X 0,Y 457.214,Z 538.815,A -85,B 0,C 180,E1 -8387.55,E2 -8387.55} C_VEL
LIN {X 0,Y 457.744,Z 524.756,A -85,B 0,C 180,E1 -8388.216,E2 -8388.216} C_VEL
LIN {X 0,Y 455.286,Z 510.21,A -85,B 0,C 180,E1 -8388.819,E2 -8388.819} C_VEL
LIN {X 0,Y 453.084,Z 498.662,A -85,B 0,C 180,E1 -8389.187,E2 -8389.187} C_VEL
LIN {X 0,Y 453.353,Z 490.291,A -85,B 0,C 180,E1 -8392.321,E2 -8392.321} C_VEL
LIN {X 0,Y 453.743,Z 481.472,A -85,B 0,C 180,E1 -8395.701,E2 -8395.701} C_VEL
LIN {X 0,Y 454.136,Z 472.678,A -85,B 0,C 180,E1 -8399.174,E2 -8399.174} C_VEL
LIN {X 0,Y 454.585,Z 465.17,A -85,B 0,C 180,E1 -8402.233,E2 -8402.233} C_VEL
LIN {X 0,Y 455.056,Z 457.584,A -85,B 0,C 180,E1 -8405.44,E2 -8405.44} C_VEL
LIN {X 0,Y 455.461,Z 451.468,A -85,B 0,C 180,E1 -8408.113,E2 -8408.113} C_VEL
LIN {X 0,Y 455.372,Z 448.47,A -85,B 0,C 180,E1 -8409.495,E2 -8409.495} C_VEL
LIN {X 0,Y 454.529,Z 443.161,A -85,B 0,C 180,E1 -8412.082,E2 -8412.082} C_VEL
LIN {X 0,Y 453.507,Z 437.622,A -85,B 0,C 180,E1 -8414.979,E2 -8414.979} C_VEL
LIN {X 0,Y 453.489,Z 437.621,A -85,B 0,C 180,E1 -8418.21,E2 -8418.21} C_VEL
LIN {X 0,Y 453.511,Z 437.621,A -85,B 0,C 180,E1 -8420.79,E2 -8420.79} C_VEL
LIN {X 0,Y 453.451,Z 437.625,A -85,B 0,C 180,E1 -8423.917,E2 -8423.917} C_VEL
LIN {X 0,Y 453.478,Z 437.625,A -85,B 0,C 180,E1 -8427.151,E2 -8427.151} C_VEL
LIN {X 0,Y 453.509,Z 437.62,A -85,B 0,C 180,E1 -8430.271,E2 -8430.271} C_VEL
LIN {X 0,Y 453.508,Z 437.62,A -85,B 0,C 180,E1 -8433.294,E2 -8433.294} C_VEL
LIN {X 0,Y 453.497,Z 437.62,A -85,B 0,C 180,E1 -8436.239,E2 -8436.239} C_VEL
LIN {X 0,Y 453.477,Z 437.624,A -85,B 0,C 180,E1 -8439.117,E2 -8439.117} C_VEL
LIN {X 0,Y 453.505,Z 437.618,A -85,B 0,C 180,E1 -8441.944,E2 -8441.944} C_VEL
LIN {X 0,Y 453.533,Z 437.617,A -85,B 0,C 180,E1 -8444.726,E2 -8444.726} C_VEL
LIN {X 0,Y 453.555,Z 437.615,A -85,B 0,C 180,E1 -8448.379,E2 -8448.379} C_VEL
LIN {X 0,Y 453.645,Z 437.602,A -85,B 0,C 180,E1 -8451.985,E2 -8451.985} C_VEL
LIN {X 0,Y 453.666,Z 437.602,A -85,B 0,C 180,E1 -8454.667,E2 -8454.667} C_VEL
LIN {X 0,Y 453.76,Z 437.589,A -85,B 0,C 180,E1 -8457.337,E2 -8457.337} C_VEL
LIN {X 0,Y 453.816,Z 437.58,A -85,B 0,C 180,E1 -8460,E2 -8460} C_VEL
LIN {X 0,Y 453.761,Z 437.589,A -85,B 0,C 180,E1 -8462.663,E2 -8462.663} C_VEL
LIN {X 0,Y 453.678,Z 437.6,A -85,B 0,C 180,E1 -8466.225,E2 -8466.225} C_VEL
LIN {X 0,Y 453.587,Z 437.61,A -85,B 0,C 180,E1 -8468.914,E2 -8468.914} C_VEL
LIN {X 0,Y 453.557,Z 437.616,A -85,B 0,C 180,E1 -8472.529,E2 -8472.529} C_VEL
LIN {X 0,Y 453.539,Z 437.616,A -85,B 0,C 180,E1 -8476.196,E2 -8476.196} C_VEL
LIN {X 0,Y 453.515,Z 437.619,A -85,B 0,C 180,E1 -8479.041,E2 -8479.041} C_VEL
LIN {X 0,Y 453.472,Z 437.624,A -85,B 0,C 180,E1 -8481.837,E2 -8481.837} C_VEL
LIN {X 0,Y 453.509,Z 437.621,A -85,B 0,C 180,E1 -8484.735,E2 -8484.735} C_VEL
LIN {X 0,Y 453.527,Z 437.62,A -85,B 0,C 180,E1 -8487.96,E2 -8487.96} C_VEL
LIN {X 0,Y 453.463,Z 437.624,A -85,B 0,C 180,E1 -8491.526,E2 -8491.526} C_VEL
LIN {X 0,Y 453.485,Z 437.623,A -85,B 0,C 180,E1 -8494.778,E2 -8494.778} C_VEL
LIN {X 0,Y 453.47,Z 437.625,A -85,B 0,C 180,E1 -8498.311,E2 -8498.311} C_VEL
LIN {X 0,Y 453.492,Z 437.621,A -85,B 0,C 180,E1 -8500.61,E2 -8500.61} C_VEL
LIN {X 0,Y 453.461,Z 437.626,A -85,B 0,C 180,E1 -8503.246,E2 -8503.246} C_VEL
LIN {X 0,Y 453.464,Z 437.628,A -85,B 0,C 180,E1 -8505.78,E2 -8505.78} C_VEL
LIN {X 0,Y 453.515,Z 437.618,A -85,B 0,C 180,E1 -8509.406,E2 -8509.406} C_VEL
LIN {X 0,Y 453.476,Z 437.625,A -85,B 0,C 180,E1 -8512.223,E2 -8512.223} C_VEL
LIN {X 0,Y 453.49,Z 437.622,A -85,B 0,C 180,E1 -8515.223,E2 -8515.223} C_VEL
LIN {X 0,Y 453.469,Z 437.623,A -85,B 0,C 180,E1 -8518.475,E2 -8518.475} C_VEL
LIN {X 0,Y 453.517,Z 437.619,A -85,B 0,C 180,E1 -8521.289,E2 -8521.289} C_VEL
LIN {X 0,Y 453.526,Z 437.617,A -85,B 0,C 180,E1 -8524.285,E2 -8524.285} C_VEL
LIN {X 0,Y 453.482,Z 437.622,A -85,B 0,C 180,E1 -8527.205,E2 -8527.205} C_VEL
LIN {X 0,Y 453.508,Z 437.621,A -85,B 0,C 180,E1 -8530.067,E2 -8530.067} C_VEL
LIN {X 0,Y 453.509,Z 437.618,A -85,B 0,C 180,E1 -8532.876,E2 -8532.876} C_VEL
LIN {X 0,Y 453.517,Z 437.62,A -85,B 0,C 180,E1 -8535.644,E2 -8535.644} C_VEL
LIN {X 0,Y 453.563,Z 437.613,A -85,B 0,C 180,E1 -8538.379,E2 -8538.379} C_VEL
LIN {X 0,Y 453.595,Z 437.609,A -85,B 0,C 180,E1 -8541.087,E2 -8541.087} C_VEL
LIN {X 0,Y 453.599,Z 437.608,A -85,B 0,C 180,E1 -8543.098,E2 -8543.098} C_VEL
LIN {X 0,Y 452.929,Z 437.693,A -85,B 0,C 180,E1 -8543.839,E2 -8543.839} C_VEL
LIN {X 0,Y 449.997,Z 438.057,A -85,B 0,C 180,E1 -8545.041,E2 -8545.041} C_VEL
LIN {X 0,Y 447.581,Z 438.357,A -85,B 0,C 180,E1 -8546.011,E2 -8546.011} C_VEL
LIN {X 0,Y 446.648,Z 438.474,A -85,B 0,C 180,E1 -8546.762,E2 -8546.762} C_VEL
LIN {X 0,Y 446.629,Z 438.476,A -85,B 0,C 180,E1 -8547.015,E2 -8547.015} C_VEL
LIN {X 0,Y 446.797,Z 438.454,A -85,B 0,C 180,E1 -8550,E2 -8550} C_VEL
LIN {X 0,Y 446.695,Z 438.469,A -85,B 0,C 180,E1 -8552.705,E2 -8552.705} C_VEL
LIN {X 0,Y 446.646,Z 438.474,A -85,B 0,C 180,E1 -8556.324,E2 -8556.324} C_VEL
LIN {X 0,Y 446.538,Z 438.489,A -85,B 0,C 180,E1 -8559.055,E2 -8559.055} C_VEL
LIN {X 0,Y 446.525,Z 438.489,A -85,B 0,C 180,E1 -8562.729,E2 -8562.729} C_VEL
LIN {X 0,Y 446.499,Z 438.492,A -85,B 0,C 180,E1 -8566.227,E2 -8566.227} C_VEL
LIN {X 0,Y 446.472,Z 438.497,A -85,B 0,C 180,E1 -8569.303,E2 -8569.303} C_VEL
LIN {X 0,Y 446.421,Z 438.501,A -85,B 0,C 180,E1 -8572.199,E2 -8572.199} C_VEL
LIN {X 0,Y 446.46,Z 438.498,A -85,B 0,C 180,E1 -8575.152,E2 -8575.152} C_VEL
LIN {X 0,Y 446.486,Z 438.493,A -85,B 0,C 180,E1 -8578.178,E2 -8578.178} C_VEL
LIN {X 0,Y 446.415,Z 438.504,A -85,B 0,C 180,E1 -8581.3,E2 -8581.3} C_VEL
LIN {X 0,Y 446.423,Z 438.503,A -85,B 0,C 180,E1 -8583.449,E2 -8583.449} C_VEL
LIN {X 0,Y 446.246,Z 438.526,A -85,B 0,C 180,E1 -8585.641,E2 -8585.641} C_VEL
LIN {X 0,Y 445.84,Z 438.579,A -85,B 0,C 180,E1 -8589.089,E2 -8589.089} C_VEL
LIN {X 0,Y 445.779,Z 439.198,A -85,B 0,C 180,E1 -8590.269,E2 -8590.269} C_VEL
LIN {X 0,Y 445.702,Z 442.144,A -85,B 0,C 180,E1 -8593.502,E2 -8593.502} C_VEL
LIN {X 0,Y 445.652,Z 444.915,A -85,B 0,C 180,E1 -8596.503,E2 -8596.503} C_VEL
LIN {X 0,Y 445.561,Z 447.934,A -85,B 0,C 180,E1 -8599.706,E2 -8599.706} C_VEL
LIN {X 0,Y 445.58,Z 450.827,A -85,B 0,C 180,E1 -8602.639,E2 -8602.639} C_VEL
LIN {X 0,Y 449.724,Z 465.796,A -85,B 0,C 180,E1 -8603.25,E2 -8603.25} C_VEL
LIN {X 0,Y 451.336,Z 472.357,A -85,B 0,C 180,E1 -8603.574,E2 -8603.574} C_VEL
LIN {X 0,Y 450.895,Z 486.252,A -85,B 0,C 180,E1 -8604.24,E2 -8604.24} C_VEL
LIN {X 0,Y 450.207,Z 498.498,A -85,B 0,C 180,E1 -8604.992,E2 -8604.992} C_VEL
LIN {X 0,Y 449.465,Z 511.123,A -85,B 0,C 180,E1 -8605.967,E2 -8605.967} C_VEL
LIN {X 0,Y 448.706,Z 522.319,A -85,B 0,C 180,E1 -8607.024,E2 -8607.024} C_VEL
LIN {X 0,Y 447.965,Z 533.359,A -85,B 0,C 180,E1 -8608.293,E2 -8608.293} C_VEL
LIN {X 0,Y 447.366,Z 542.672,A -85,B 0,C 180,E1 -8609.586,E2 -8609.586} C_VEL
LIN {X 0,Y 446.699,Z 551.659,A -85,B 0,C 180,E1 -8611.092,E2 -8611.092} C_VEL
LIN {X 0,Y 446.316,Z 558.878,A -85,B 0,C 180,E1 -8612.574,E2 -8612.574} C_VEL
LIN {X 0,Y 445.916,Z 565.867,A -85,B 0,C 180,E1 -8614.363,E2 -8614.363} C_VEL
LIN {X 0,Y 445.659,Z 571.17,A -85,B 0,C 180,E1 -8616.154,E2 -8616.154} C_VEL
LIN {X 0,Y 445.486,Z 574.641,A -85,B 0,C 180,E1 -8617.751,E2 -8617.751} C_VEL
LIN {X 0,Y 445.442,Z 576.185,A -85,B 0,C 180,E1 -8618.722,E2 -8618.722} C_VEL
LIN {X 0,Y 445.338,Z 578.095,A -85,B 0,C 180,E1 -8620.646,E2 -8620.646} C_VEL
LIN {X 0,Y 445.352,Z 578.486,A -85,B 0,C 180,E1 -8621.602,E2 -8621.602} C_VEL
LIN {X 0,Y 445.33,Z 578.176,A -85,B 0,C 180,E1 -8623.497,E2 -8623.497} C_VEL
LIN {X 0,Y 445.415,Z 576.428,A -85,B 0,C 180,E1 -8625.377,E2 -8625.377} C_VEL
LIN {X 0,Y 445.608,Z 573.221,A -85,B 0,C 180,E1 -8627.244,E2 -8627.244} C_VEL
LIN {X 0,Y 445.866,Z 568.462,A -85,B 0,C 180,E1 -8629.097,E2 -8629.097} C_VEL
LIN {X 0,Y 446.122,Z 563.863,A -85,B 0,C 180,E1 -8630.479,E2 -8630.479} C_VEL
LIN {X 0,Y 446.439,Z 558.208,A -85,B 0,C 180,E1 -8631.855,E2 -8631.855} C_VEL
LIN {X 0,Y 447.08,Z 550.145,A -85,B 0,C 180,E1 -8633.456,E2 -8633.456} C_VEL
LIN {X 0,Y 447.603,Z 541.769,A -85,B 0,C 180,E1 -8634.82,E2 -8634.82} C_VEL
LIN {X 0,Y 448.314,Z 531.637,A -85,B 0,C 180,E1 -8636.18,E2 -8636.18} C_VEL
LIN {X 0,Y 449.14,Z 520.357,A -85,B 0,C 180,E1 -8637.421,E2 -8637.421} C_VEL
LIN {X 0,Y 449.935,Z 508.267,A -85,B 0,C 180,E1 -8638.514,E2 -8638.514} C_VEL
LIN {X 0,Y 450.714,Z 495.579,A -85,B 0,C 180,E1 -8639.438,E2 -8639.438} C_VEL
LIN {X 0,Y 451.422,Z 482.752,A -85,B 0,C 180,E1 -8640.176,E2 -8640.176} C_VEL
LIN {X 0,Y 451.677,Z 472.836,A -85,B 0,C 180,E1 -8640.633,E2 -8640.633} C_VEL
LIN {X 0,Y 447.973,Z 459.844,A -85,B 0,C 180,E1 -8641.291,E2 -8641.291} C_VEL
LIN {X 0,Y 445.777,Z 453.056,A -85,B 0,C 180,E1 -8641.589,E2 -8641.589} C_VEL
LIN {X 0,Y 446.114,Z 450.646,A -85,B 0,C 180,E1 -8644.518,E2 -8644.518} C_VEL
LIN {X 0,Y 446.173,Z 448.524,A -85,B 0,C 180,E1 -8647.239,E2 -8647.239} C_VEL
LIN {X 0,Y 446.149,Z 446.483,A -85,B 0,C 180,E1 -8649.978,E2 -8649.978} C_VEL
LIN {X 0,Y 446.288,Z 444.463,A -85,B 0,C 180,E1 -8652.736,E2 -8652.736} C_VEL
LIN {X 0,Y 446.406,Z 442.107,A -85,B 0,C 180,E1 -8656.191,E2 -8656.191} C_VEL
LIN {X 0,Y 446.553,Z 440.144,A -85,B 0,C 180,E1 -8659.299,E2 -8659.299} C_VEL
LIN {X 0,Y 446.41,Z 438.53,A -85,B 0,C 180,E1 -8662.2,E2 -8662.2} C_VEL
LIN {X 0,Y 446.452,Z 438.5,A -85,B 0,C 180,E1 -8665.152,E2 -8665.152} C_VEL
LIN {X 0,Y 446.479,Z 438.497,A -85,B 0,C 180,E1 -8668.179,E2 -8668.179} C_VEL
LIN {X 0,Y 446.415,Z 438.504,A -85,B 0,C 180,E1 -8671.3,E2 -8671.3} C_VEL
LIN {X 0,Y 446.426,Z 438.503,A -85,B 0,C 180,E1 -8674.523,E2 -8674.523} C_VEL
LIN {X 0,Y 446.432,Z 438.503,A -85,B 0,C 180,E1 -8678.083,E2 -8678.083} C_VEL
LIN {X 0,Y 446.48,Z 438.644,A -85,B 0,C 180,E1 -8680.927,E2 -8680.927} C_VEL
LIN {X 0,Y 446.955,Z 441.213,A -85,B 0,C 180,E1 -8683.778,E2 -8683.778} C_VEL
LIN {X 0,Y 447.561,Z 444.943,A -85,B 0,C 180,E1 -8686.917,E2 -8686.917} C_VEL
LIN {X 0,Y 448.077,Z 447.696,A -85,B 0,C 180,E1 -8688.84,E2 -8688.84} C_VEL
LIN {X 0,Y 448.435,Z 451.48,A -85,B 0,C 180,E1 -8691.18,E2 -8691.18} C_VEL
LIN {X 0,Y 448.201,Z 455.048,A -85,B 0,C 180,E1 -8693.102,E2 -8693.102} C_VEL
LIN {X 0,Y 447.506,Z 462.369,A -85,B 0,C 180,E1 -8696.656,E2 -8696.656} C_VEL
LIN {X 0,Y 447.063,Z 469.523,A -85,B 0,C 180,E1 -8699.839,E2 -8699.839} C_VEL
LIN {X 0,Y 446.636,Z 476.753,A -85,B 0,C 180,E1 -8702.85,E2 -8702.85} C_VEL
LIN {X 0,Y 446.285,Z 484.652,A -85,B 0,C 180,E1 -8705.976,E2 -8705.976} C_VEL
LIN {X 0,Y 446.056,Z 491.942,A -85,B 0,C 180,E1 -8708.754,E2 -8708.754} C_VEL
LIN {X 0,Y 445.947,Z 496.271,A -85,B 0,C 180,E1 -8710.37,E2 -8710.37} C_VEL
LIN {X 0,Y 448.897,Z 512.219,A -85,B 0,C 180,E1 -8710.951,E2 -8710.951} C_VEL
LIN {X 0,Y 450.925,Z 527.34,A -85,B 0,C 180,E1 -8711.657,E2 -8711.657} C_VEL
LIN {X 0,Y 450.174,Z 541.044,A -85,B 0,C 180,E1 -8712.377,E2 -8712.377} C_VEL
LIN {X 0,Y 449.328,Z 554.759,A -85,B 0,C 180,E1 -8713.298,E2 -8713.298} C_VEL
LIN {X 0,Y 448.482,Z 566.924,A -85,B 0,C 180,E1 -8714.317,E2 -8714.317} C_VEL
LIN {X 0,Y 447.721,Z 578.089,A -85,B 0,C 180,E1 -8715.454,E2 -8715.454} C_VEL
LIN {X 0,Y 447.051,Z 589.162,A -85,B 0,C 180,E1 -8716.824,E2 -8716.824} C_VEL
LIN {X 0,Y 446.509,Z 598.338,A -85,B 0,C 180,E1 -8718.193,E2 -8718.193} C_VEL
LIN {X 0,Y 446.045,Z 607.151,A -85,B 0,C 180,E1 -8719.79,E2 -8719.79} C_VEL
LIN {X 0,Y 445.742,Z 614.278,A -85,B 0,C 180,E1 -8721.386,E2 -8721.386} C_VEL
LIN {X 0,Y 445.575,Z 619.219,A -85,B 0,C 180,E1 -8722.751,E2 -8722.751} C_VEL
LIN {X 0,Y 445.513,Z 622.676,A -85,B 0,C 180,E1 -8723.904,E2 -8723.904} C_VEL
LIN {X 0,Y 445.413,Z 626.314,A -85,B 0,C 180,E1 -8725.475,E2 -8725.475} C_VEL
LIN {X 0,Y 445.454,Z 629.167,A -85,B 0,C 180,E1 -8727.287,E2 -8727.287} C_VEL
LIN {X 0,Y 445.424,Z 630.599,A -85,B 0,C 180,E1 -8729.096,E2 -8729.096} C_VEL
LIN {X 0,Y 445.424,Z 630.639,A -85,B 0,C 180,E1 -8730.904,E2 -8730.904} C_VEL
LIN {X 0,Y 445.451,Z 629.295,A -85,B 0,C 180,E1 -8732.713,E2 -8732.713} C_VEL
LIN {X 0,Y 445.408,Z 626.54,A -85,B 0,C 180,E1 -8734.525,E2 -8734.525} C_VEL
LIN {X 0,Y 445.488,Z 623.065,A -85,B 0,C 180,E1 -8736.067,E2 -8736.067} C_VEL
LIN {X 0,Y 445.58,Z 618.107,A -85,B 0,C 180,E1 -8737.705,E2 -8737.705} C_VEL
LIN {X 0,Y 445.807,Z 612.903,A -85,B 0,C 180,E1 -8739.07,E2 -8739.07} C_VEL
LIN {X 0,Y 446.176,Z 605.442,A -85,B 0,C 180,E1 -8740.666,E2 -8740.666} C_VEL
LIN {X 0,Y 446.641,Z 597.627,A -85,B 0,C 180,E1 -8742.034,E2 -8742.034} C_VEL
LIN {X 0,Y 447.16,Z 588.416,A -85,B 0,C 180,E1 -8743.381,E2 -8743.381} C_VEL
LIN {X 0,Y 447.879,Z 577.888,A -85,B 0,C 180,E1 -8744.657,E2 -8744.657} C_VEL
LIN {X 0,Y 448.654,Z 566.508,A -85,B 0,C 180,E1 -8745.793,E2 -8745.793} C_VEL
LIN {X 0,Y 449.464,Z 553.996,A -85,B 0,C 180,E1 -8746.814,E2 -8746.814} C_VEL
LIN {X 0,Y 450.282,Z 540.915,A -85,B 0,C 180,E1 -8747.666,E2 -8747.666} C_VEL
LIN {X 0,Y 450.928,Z 527.662,A -85,B 0,C 180,E1 -8748.34,E2 -8748.34} C_VEL
LIN {X 0,Y 450.153,Z 521.318,A -85,B 0,C 180,E1 -8748.642,E2 -8748.642} C_VEL
LIN {X 0,Y 447.699,Z 506.913,A -85,B 0,C 180,E1 -8749.216,E2 -8749.216} C_VEL
LIN {X 0,Y 446.021,Z 498.294,A -85,B 0,C 180,E1 -8749.502,E2 -8749.502} C_VEL
LIN {X 0,Y 446.331,Z 489.955,A -85,B 0,C 180,E1 -8752.692,E2 -8752.692} C_VEL
LIN {X 0,Y 446.759,Z 480.798,A -85,B 0,C 180,E1 -8756.276,E2 -8756.276} C_VEL
LIN {X 0,Y 447.186,Z 472.39,A -85,B 0,C 180,E1 -8759.673,E2 -8759.673} C_VEL
LIN {X 0,Y 447.665,Z 464.892,A -85,B 0,C 180,E1 -8762.794,E2 -8762.794} C_VEL
LIN {X 0,Y 448.156,Z 457.423,A -85,B 0,C 180,E1 -8766.02,E2 -8766.02} C_VEL
LIN {X 0,Y 448.494,Z 452.088,A -85,B 0,C 180,E1 -8768.417,E2 -8768.417} C_VEL
LIN {X 0,Y 448.124,Z 447.577,A -85,B 0,C 180,E1 -8770.559,E2 -8770.559} C_VEL
LIN {X 0,Y 446.943,Z 441.272,A -85,B 0,C 180,E1 -8773.778,E2 -8773.778} C_VEL
LIN {X 0,Y 446.464,Z 438.499,A -85,B 0,C 180,E1 -8775.267,E2 -8775.267} C_VEL
LIN {X 0,Y 446.433,Z 438.5,A -85,B 0,C 180,E1 -8778.61,E2 -8778.61} C_VEL
LIN {X 0,Y 446.455,Z 438.499,A -85,B 0,C 180,E1 -8780.974,E2 -8780.974} C_VEL
LIN {X 0,Y 446.416,Z 438.502,A -85,B 0,C 180,E1 -8784.374,E2 -8784.374} C_VEL
LIN {X 0,Y 446.425,Z 438.501,A -85,B 0,C 180,E1 -8787.639,E2 -8787.639} C_VEL
LIN {X 0,Y 446.464,Z 438.498,A -85,B 0,C 180,E1 -8790.792,E2 -8790.792} C_VEL
LIN {X 0,Y 446.472,Z 438.495,A -85,B 0,C 180,E1 -8793.848,E2 -8793.848} C_VEL
LIN {X 0,Y 446.424,Z 438.504,A -85,B 0,C 180,E1 -8796.823,E2 -8796.823} C_VEL
LIN {X 0,Y 446.438,Z 438.5,A -85,B 0,C 180,E1 -8799.737,E2 -8799.737} C_VEL
LIN {X 0,Y 446.457,Z 438.5,A -85,B 0,C 180,E1 -8802.597,E2 -8802.597} C_VEL
LIN {X 0,Y 446.463,Z 438.497,A -85,B 0,C 180,E1 -8805.412,E2 -8805.412} C_VEL
LIN {X 0,Y 446.512,Z 438.492,A -85,B 0,C 180,E1 -8808.193,E2 -8808.193} C_VEL
LIN {X 0,Y 446.594,Z 438.48,A -85,B 0,C 180,E1 -8811.858,E2 -8811.858} C_VEL
LIN {X 0,Y 446.64,Z 438.476,A -85,B 0,C 180,E1 -8814.583,E2 -8814.583} C_VEL
LIN {X 0,Y 446.704,Z 438.468,A -85,B 0,C 180,E1 -8817.295,E2 -8817.295} C_VEL
LIN {X 0,Y 446.787,Z 438.456,A -85,B 0,C 180,E1 -8820,E2 -8820} C_VEL
LIN {X 0,Y 446.704,Z 438.469,A -85,B 0,C 180,E1 -8822.705,E2 -8822.705} C_VEL
LIN {X 0,Y 446.646,Z 438.476,A -85,B 0,C 180,E1 -8826.324,E2 -8826.324} C_VEL
LIN {X 0,Y 446.532,Z 438.488,A -85,B 0,C 180,E1 -8829.056,E2 -8829.056} C_VEL
LIN {X 0,Y 446.515,Z 438.492,A -85,B 0,C 180,E1 -8832.73,E2 -8832.73} C_VEL
LIN {X 0,Y 446.49,Z 438.494,A -85,B 0,C 180,E1 -8836.228,E2 -8836.228} C_VEL
LIN {X 0,Y 446.464,Z 438.496,A -85,B 0,C 180,E1 -8839.304,E2 -8839.304} C_VEL
LIN {X 0,Y 446.414,Z 438.505,A -85,B 0,C 180,E1 -8842.2,E2 -8842.2} C_VEL
LIN {X 0,Y 446.453,Z 438.498,A -85,B 0,C 180,E1 -8845.153,E2 -8845.153} C_VEL
LIN {X 0,Y 446.48,Z 438.497,A -85,B 0,C 180,E1 -8848.179,E2 -8848.179} C_VEL
LIN {X 0,Y 446.416,Z 438.503,A -85,B 0,C 180,E1 -8851.776,E2 -8851.776} C_VEL
LIN {X 0,Y 446.427,Z 438.504,A -85,B 0,C 180,E1 -8854.524,E2 -8854.524} C_VEL
LIN {X 0,Y 446.427,Z 438.502,A -85,B 0,C 180,E1 -8858.082,E2 -8858.082} C_VEL
LIN {X 0,Y 446.425,Z 438.5,A -85,B 0,C 180,E1 -8860.918,E2 -8860.918} C_VEL
LIN {X 0,Y 446.421,Z 438.503,A -85,B 0,C 180,E1 -8863.844,E2 -8863.844} C_VEL
LIN {X 0,Y 446.398,Z 438.506,A -85,B 0,C 180,E1 -8866.404,E2 -8866.404} C_VEL
LIN {X 0,Y 446.467,Z 438.499,A -85,B 0,C 180,E1 -8869.806,E2 -8869.806} C_VEL
LIN {X 0,Y 446.433,Z 438.502,A -85,B 0,C 180,E1 -8872.124,E2 -8872.124} C_VEL
LIN {X 0,Y 446.431,Z 438.503,A -85,B 0,C 180,E1 -8875.478,E2 -8875.478} C_VEL
LIN {X 0,Y 446.42,Z 438.5,A -85,B 0,C 180,E1 -8878.701,E2 -8878.701} C_VEL
LIN {X 0,Y 446.486,Z 438.496,A -85,B 0,C 180,E1 -8881.822,E2 -8881.822} C_VEL
LIN {X 0,Y 446.459,Z 438.497,A -85,B 0,C 180,E1 -8884.848,E2 -8884.848} C_VEL
LIN {X 0,Y 446.451,Z 438.498,A -85,B 0,C 180,E1 -8888.246,E2 -8888.246} C_VEL
LIN {X 0,Y 446.46,Z 438.5,A -85,B 0,C 180,E1 -8891.65,E2 -8891.65} C_VEL
LIN {X 0,Y 446.511,Z 438.491,A -85,B 0,C 180,E1 -8894.48,E2 -8894.48} C_VEL
LIN {X 0,Y 446.521,Z 438.49,A -85,B 0,C 180,E1 -8898.193,E2 -8898.193} C_VEL
LIN {X 0,Y 446.541,Z 438.487,A -85,B 0,C 180,E1 -8900.945,E2 -8900.945} C_VEL
LIN {X 0,Y 446.623,Z 438.478,A -85,B 0,C 180,E1 -8903.676,E2 -8903.676} C_VEL
LIN {X 0,Y 446.629,Z 438.476,A -85,B 0,C 180,E1 -8907.015,E2 -8907.015} C_VEL
LIN {X 0,Y 446.427,Z 438.504,A -85,B 0,C 180,E1 -8907.519,E2 -8907.519} C_VEL
LIN {X 0,Y 445.16,Z 438.664,A -85,B 0,C 180,E1 -8908.262,E2 -8908.262} C_VEL
LIN {X 0,Y 440.79,Z 439.208,A -85,B 0,C 180,E1 -8909.978,E2 -8909.978} C_VEL
LIN {X 0,Y 439.704,Z 439.34,A -85,B 0,C 180,E1 -8910.741,E2 -8910.741} C_VEL
LIN {X 0,Y 439.613,Z 439.35,A -85,B 0,C 180,E1 -8911,E2 -8911} C_VEL
LIN {X 0,Y 439.645,Z 439.347,A -85,B 0,C 180,E1 -8912.749,E2 -8912.749} C_VEL
LIN {X 0,Y 439.617,Z 439.349,A -85,B 0,C 180,E1 -8916.425,E2 -8916.425} C_VEL
LIN {X 0,Y 439.501,Z 439.367,A -85,B 0,C 180,E1 -8919.201,E2 -8919.201} C_VEL
LIN {X 0,Y 439.469,Z 439.369,A -85,B 0,C 180,E1 -8922.937,E2 -8922.937} C_VEL
LIN {X 0,Y 439.45,Z 439.37,A -85,B 0,C 180,E1 -8926.348,E2 -8926.348} C_VEL
LIN {X 0,Y 439.405,Z 439.376,A -85,B 0,C 180,E1 -8929.626,E2 -8929.626} C_VEL
LIN {X 0,Y 439.368,Z 439.38,A -85,B 0,C 180,E1 -8932.575,E2 -8932.575} C_VEL
LIN {X 0,Y 439.407,Z 439.377,A -85,B 0,C 180,E1 -8935.584,E2 -8935.584} C_VEL
LIN {X 0,Y 439.419,Z 439.376,A -85,B 0,C 180,E1 -8938.673,E2 -8938.673} C_VEL
LIN {X 0,Y 439.366,Z 439.379,A -85,B 0,C 180,E1 -8942.029,E2 -8942.029} C_VEL
LIN {X 0,Y 439.285,Z 439.394,A -85,B 0,C 180,E1 -8945.166,E2 -8945.166} C_VEL
LIN {X 0,Y 438.879,Z 439.444,A -85,B 0,C 180,E1 -8948.31,E2 -8948.31} C_VEL
LIN {X 0,Y 438.706,Z 439.529,A -85,B 0,C 180,E1 -8949.85,E2 -8949.85} C_VEL
LIN {X 0,Y 438.667,Z 441.922,A -85,B 0,C 180,E1 -8952.525,E2 -8952.525} C_VEL
LIN {X 0,Y 438.613,Z 444.351,A -85,B 0,C 180,E1 -8955.168,E2 -8955.168} C_VEL
LIN {X 0,Y 438.557,Z 446.694,A -85,B 0,C 180,E1 -8957.696,E2 -8957.696} C_VEL
LIN {X 0,Y 438.485,Z 450.096,A -85,B 0,C 180,E1 -8961.311,E2 -8961.311} C_VEL
LIN {X 0,Y 438.5,Z 451.158,A -85,B 0,C 180,E1 -8962.336,E2 -8962.336} C_VEL
LIN {X 0,Y 442.643,Z 466.104,A -85,B 0,C 180,E1 -8962.962,E2 -8962.962} C_VEL
LIN {X 0,Y 444.583,Z 473.807,A -85,B 0,C 180,E1 -8963.354,E2 -8963.354} C_VEL
LIN {X 0,Y 444.005,Z 488.261,A -85,B 0,C 180,E1 -8964.081,E2 -8964.081} C_VEL
LIN {X 0,Y 443.247,Z 501.138,A -85,B 0,C 180,E1 -8964.916,E2 -8964.916} C_VEL
LIN {X 0,Y 442.51,Z 512.709,A -85,B 0,C 180,E1 -8965.849,E2 -8965.849} C_VEL
LIN {X 0,Y 441.721,Z 524.219,A -85,B 0,C 180,E1 -8966.979,E2 -8966.979} C_VEL
LIN {X 0,Y 440.958,Z 535.01,A -85,B 0,C 180,E1 -8968.267,E2 -8968.267} C_VEL
LIN {X 0,Y 440.318,Z 544.362,A -85,B 0,C 180,E1 -8969.616,E2 -8969.616} C_VEL
LIN {X 0,Y 439.657,Z 552.8,A -85,B 0,C 180,E1 -8971.082,E2 -8971.082} C_VEL
LIN {X 0,Y 439.244,Z 560.003,A -85,B 0,C 180,E1 -8972.612,E2 -8972.612} C_VEL
LIN {X 0,Y 438.85,Z 566.668,A -85,B 0,C 180,E1 -8974.38,E2 -8974.38} C_VEL
LIN {X 0,Y 438.606,Z 571.304,A -85,B 0,C 180,E1 -8975.969,E2 -8975.969} C_VEL
LIN {X 0,Y 438.423,Z 574.411,A -85,B 0,C 180,E1 -8977.373,E2 -8977.373} C_VEL
LIN {X 0,Y 438.396,Z 576.183,A -85,B 0,C 180,E1 -8978.402,E2 -8978.402} C_VEL
LIN {X 0,Y 438.264,Z 578.33,A -85,B 0,C 180,E1 -8980.32,E2 -8980.32} C_VEL
LIN {X 0,Y 438.29,Z 578.837,A -85,B 0,C 180,E1 -8981.294,E2 -8981.294} C_VEL
LIN {X 0,Y 438.232,Z 578.753,A -85,B 0,C 180,E1 -8983.221,E2 -8983.221} C_VEL
LIN {X 0,Y 438.32,Z 577.223,A -85,B 0,C 180,E1 -8985.135,E2 -8985.135} C_VEL
LIN {X 0,Y 438.503,Z 574.255,A -85,B 0,C 180,E1 -8987.033,E2 -8987.033} C_VEL
LIN {X 0,Y 438.768,Z 569.799,A -85,B 0,C 180,E1 -8988.918,E2 -8988.918} C_VEL
LIN {X 0,Y 439.042,Z 565.347,A -85,B 0,C 180,E1 -8990.324,E2 -8990.324} C_VEL
LIN {X 0,Y 439.385,Z 559.924,A -85,B 0,C 180,E1 -8991.723,E2 -8991.723} C_VEL
LIN {X 0,Y 439.971,Z 552.164,A -85,B 0,C 180,E1 -8993.349,E2 -8993.349} C_VEL
LIN {X 0,Y 440.553,Z 544.103,A -85,B 0,C 180,E1 -8994.737,E2 -8994.737} C_VEL
LIN {X 0,Y 441.292,Z 534.433,A -85,B 0,C 180,E1 -8996.119,E2 -8996.119} C_VEL
LIN {X 0,Y 442.131,Z 523.732,A -85,B 0,C 180,E1 -8997.38,E2 -8997.38} C_VEL
LIN {X 0,Y 443.021,Z 511.742,A -85,B 0,C 180,E1 -8998.537,E2 -8998.537} C_VEL
LIN {X 0,Y 443.832,Z 498.733,A -85,B 0,C 180,E1 -8999.546,E2 -8999.546} C_VEL
LIN {X 0,Y 444.623,Z 485.051,A -85,B 0,C 180,E1 -9000.38,E2 -9000.38} C_VEL
LIN {X 0,Y 444.974,Z 474.26,A -85,B 0,C 180,E1 -9000.905,E2 -9000.905} C_VEL
LIN {X 0,Y 441.037,Z 460.466,A -85,B 0,C 180,E1 -9001.636,E2 -9001.636} C_VEL
LIN {X 0,Y 438.732,Z 453.586,A -85,B 0,C 180,E1 -9001.979,E2 -9001.979} C_VEL
LIN {X 0,Y 439.082,Z 451.474,A -85,B 0,C 180,E1 -9004.59,E2 -9004.59} C_VEL
LIN {X 0,Y 439.153,Z 449.347,A -85,B 0,C 180,E1 -9007.356,E2 -9007.356} C_VEL
LIN {X 0,Y 439.123,Z 447.306,A -85,B 0,C 180,E1 -9010.14,E2 -9010.14} C_VEL
LIN {X 0,Y 439.261,Z 445.339,A -85,B 0,C 180,E1 -9012.944,E2 -9012.944} C_VEL
LIN {X 0,Y 439.392,Z 443.068,A -85,B 0,C 180,E1 -9016.327,E2 -9016.327} C_VEL
LIN {X 0,Y 439.554,Z 441.218,A -85,B 0,C 180,E1 -9019.381,E2 -9019.381} C_VEL
LIN {X 0,Y 439.389,Z 439.551,A -85,B 0,C 180,E1 -9022.574,E2 -9022.574} C_VEL
LIN {X 0,Y 439.4,Z 439.378,A -85,B 0,C 180,E1 -9025.585,E2 -9025.585} C_VEL
LIN {X 0,Y 439.42,Z 439.376,A -85,B 0,C 180,E1 -9028.673,E2 -9028.673} C_VEL
LIN {X 0,Y 439.369,Z 439.382,A -85,B 0,C 180,E1 -9031.861,E2 -9031.861} C_VEL
LIN {X 0,Y 439.396,Z 439.379,A -85,B 0,C 180,E1 -9035.156,E2 -9035.156} C_VEL
LIN {X 0,Y 439.393,Z 439.379,A -85,B 0,C 180,E1 -9038.594,E2 -9038.594} C_VEL
LIN {X 0,Y 439.434,Z 439.457,A -85,B 0,C 180,E1 -9039.855,E2 -9039.855} C_VEL
LIN {X 0,Y 439.958,Z 442.356,A -85,B 0,C 180,E1 -9043.385,E2 -9043.385} C_VEL
LIN {X 0,Y 440.596,Z 446.18,A -85,B 0,C 180,E1 -9046.695,E2 -9046.695} C_VEL
LIN {X 0,Y 441.193,Z 449.704,A -85,B 0,C 180,E1 -9049.224,E2 -9049.224} C_VEL
LIN {X 0,Y 441.459,Z 453.61,A -85,B 0,C 180,E1 -9051.621,E2 -9051.621} C_VEL
LIN {X 0,Y 440.888,Z 458.846,A -85,B 0,C 180,E1 -9054.387,E2 -9054.387} C_VEL
LIN {X 0,Y 440.47,Z 464.54,A -85,B 0,C 180,E1 -9057.147,E2 -9057.147} C_VEL
LIN {X 0,Y 439.985,Z 471.638,A -85,B 0,C 180,E1 -9060.32,E2 -9060.32} C_VEL
LIN {X 0,Y 439.514,Z 479.345,A -85,B 0,C 180,E1 -9063.568,E2 -9063.568} C_VEL
LIN {X 0,Y 439.117,Z 487.722,A -85,B 0,C 180,E1 -9066.914,E2 -9066.914} C_VEL
LIN {X 0,Y 438.891,Z 495.837,A -85,B 0,C 180,E1 -9070.012,E2 -9070.012} C_VEL
LIN {X 0,Y 441.874,Z 511.237,A -85,B 0,C 180,E1 -9070.594,E2 -9070.594} C_VEL
LIN {X 0,Y 443.973,Z 526.069,A -85,B 0,C 180,E1 -9071.301,E2 -9071.301} C_VEL
LIN {X 0,Y 443.761,Z 535.257,A -85,B 0,C 180,E1 -9071.774,E2 -9071.774} C_VEL
LIN {X 0,Y 442.897,Z 548.175,A -85,B 0,C 180,E1 -9072.572,E2 -9072.572} C_VEL
LIN {X 0,Y 442,Z 561.418,A -85,B 0,C 180,E1 -9073.607,E2 -9073.607} C_VEL
LIN {X 0,Y 441.07,Z 573.409,A -85,B 0,C 180,E1 -9074.757,E2 -9074.757} C_VEL
LIN {X 0,Y 440.27,Z 585.259,A -85,B 0,C 180,E1 -9076.147,E2 -9076.147} C_VEL
LIN {X 0,Y 439.711,Z 595.354,A -85,B 0,C 180,E1 -9077.587,E2 -9077.587} C_VEL
LIN {X 0,Y 439.114,Z 604.412,A -85,B 0,C 180,E1 -9079.161,E2 -9079.161} C_VEL
LIN {X 0,Y 438.73,Z 611.973,A -85,B 0,C 180,E1 -9080.782,E2 -9080.782} C_VEL
LIN {X 0,Y 438.505,Z 617.28,A -85,B 0,C 180,E1 -9082.17,E2 -9082.17} C_VEL
LIN {X 0,Y 438.504,Z 621.555,A -85,B 0,C 180,E1 -9083.559,E2 -9083.559} C_VEL
LIN {X 0,Y 438.338,Z 625.886,A -85,B 0,C 180,E1 -9085.402,E2 -9085.402} C_VEL
LIN {X 0,Y 438.382,Z 628.745,A -85,B 0,C 180,E1 -9087.243,E2 -9087.243} C_VEL
LIN {X 0,Y 438.363,Z 630.183,A -85,B 0,C 180,E1 -9089.081,E2 -9089.081} C_VEL
LIN {X 0,Y 438.363,Z 630.224,A -85,B 0,C 180,E1 -9090.919,E2 -9090.919} C_VEL
LIN {X 0,Y 438.377,Z 628.876,A -85,B 0,C 180,E1 -9092.757,E2 -9092.757} C_VEL
LIN {X 0,Y 438.333,Z 626.115,A -85,B 0,C 180,E1 -9094.598,E2 -9094.598} C_VEL
LIN {X 0,Y 438.446,Z 621.874,A -85,B 0,C 180,E1 -9096.442,E2 -9096.442} C_VEL
LIN {X 0,Y 438.587,Z 616.024,A -85,B 0,C 180,E1 -9098.292,E2 -9098.292} C_VEL
LIN {X 0,Y 438.877,Z 609.424,A -85,B 0,C 180,E1 -9099.912,E2 -9099.912} C_VEL
LIN {X 0,Y 439.387,Z 601.235,A -85,B 0,C 180,E1 -9101.533,E2 -9101.533} C_VEL
LIN {X 0,Y 439.889,Z 592.513,A -85,B 0,C 180,E1 -9102.946,E2 -9102.946} C_VEL
LIN {X 0,Y 440.59,Z 582.282,A -85,B 0,C 180,E1 -9104.314,E2 -9104.314} C_VEL
LIN {X 0,Y 441.417,Z 570.714,A -85,B 0,C 180,E1 -9105.585,E2 -9105.585} C_VEL
LIN {X 0,Y 442.255,Z 559.241,A -85,B 0,C 180,E1 -9106.621,E2 -9106.621} C_VEL
LIN {X 0,Y 443.022,Z 546.742,A -85,B 0,C 180,E1 -9107.542,E2 -9107.542} C_VEL
LIN {X 0,Y 443.836,Z 533.567,A -85,B 0,C 180,E1 -9108.308,E2 -9108.308} C_VEL
LIN {X 0,Y 444.083,Z 527.416,A -85,B 0,C 180,E1 -9108.605,E2 -9108.605} C_VEL
LIN {X 0,Y 441.817,Z 512.978,A -85,B 0,C 180,E1 -9109.27,E2 -9109.27} C_VEL
LIN {X 0,Y 438.996,Z 497.951,A -85,B 0,C 180,E1 -9109.809,E2 -9109.809} C_VEL
LIN {X 0,Y 439.308,Z 489.589,A -85,B 0,C 180,E1 -9113.075,E2 -9113.075} C_VEL
LIN {X 0,Y 439.73,Z 481.062,A -85,B 0,C 180,E1 -9116.489,E2 -9116.489} C_VEL
LIN {X 0,Y 440.149,Z 473.33,A -85,B 0,C 180,E1 -9119.668,E2 -9119.668} C_VEL
LIN {X 0,Y 440.644,Z 465.859,A -85,B 0,C 180,E1 -9122.838,E2 -9122.838} C_VEL
LIN {X 0,Y 441.167,Z 458.397,A -85,B 0,C 180,E1 -9126.116,E2 -9126.116} C_VEL
LIN {X 0,Y 441.496,Z 452.667,A -85,B 0,C 180,E1 -9128.738,E2 -9128.738} C_VEL
LIN {X 0,Y 441.081,Z 448.461,A -85,B 0,C 180,E1 -9130.788,E2 -9130.788} C_VEL
LIN {X 0,Y 439.924,Z 442.195,A -85,B 0,C 180,E1 -9134.037,E2 -9134.037} C_VEL
LIN {X 0,Y 439.431,Z 439.374,A -85,B 0,C 180,E1 -9135.59,E2 -9135.59} C_VEL
LIN {X 0,Y 439.381,Z 439.38,A -85,B 0,C 180,E1 -9139.019,E2 -9139.019} C_VEL
LIN {X 0,Y 439.373,Z 439.382,A -85,B 0,C 180,E1 -9141.607,E2 -9141.607} C_VEL
LIN {X 0,Y 439.395,Z 439.38,A -85,B 0,C 180,E1 -9144.844,E2 -9144.844} C_VEL
LIN {X 0,Y 439.385,Z 439.376,A -85,B 0,C 180,E1 -9148.141,E2 -9148.141} C_VEL
LIN {X 0,Y 439.42,Z 439.377,A -85,B 0,C 180,E1 -9151.327,E2 -9151.327} C_VEL
LIN {X 0,Y 439.4,Z 439.378,A -85,B 0,C 180,E1 -9154.415,E2 -9154.415} C_VEL
LIN {X 0,Y 439.359,Z 439.381,A -85,B 0,C 180,E1 -9157.424,E2 -9157.424} C_VEL
LIN {X 0,Y 439.435,Z 439.373,A -85,B 0,C 180,E1 -9160.663,E2 -9160.663} C_VEL
LIN {X 0,Y 439.456,Z 439.371,A -85,B 0,C 180,E1 -9164.224,E2 -9164.224} C_VEL
LIN {X 0,Y 439.478,Z 439.367,A -85,B 0,C 180,E1 -9168.001,E2 -9168.001} C_VEL
LIN {X 0,Y 439.542,Z 439.358,A -85,B 0,C 180,E1 -9171.726,E2 -9171.726} C_VEL
LIN {X 0,Y 439.616,Z 439.351,A -85,B 0,C 180,E1 -9174.496,E2 -9174.496} C_VEL
LIN {X 0,Y 439.63,Z 439.349,A -85,B 0,C 180,E1 -9178.168,E2 -9178.168} C_VEL
LIN {X 0,Y 439.757,Z 439.331,A -85,B 0,C 180,E1 -9180,E2 -9180} C_VEL
LIN {X 0,Y 439.651,Z 439.347,A -85,B 0,C 180,E1 -9182.749,E2 -9182.749} C_VEL
LIN {X 0,Y 439.617,Z 439.351,A -85,B 0,C 180,E1 -9186.425,E2 -9186.425} C_VEL
LIN {X 0,Y 439.494,Z 439.364,A -85,B 0,C 180,E1 -9189.202,E2 -9189.202} C_VEL
LIN {X 0,Y 439.459,Z 439.369,A -85,B 0,C 180,E1 -9192.938,E2 -9192.938} C_VEL
LIN {X 0,Y 439.442,Z 439.373,A -85,B 0,C 180,E1 -9196.349,E2 -9196.349} C_VEL
LIN {X 0,Y 439.397,Z 439.377,A -85,B 0,C 180,E1 -9199.627,E2 -9199.627} C_VEL
LIN {X 0,Y 439.36,Z 439.383,A -85,B 0,C 180,E1 -9202.576,E2 -9202.576} C_VEL
LIN {X 0,Y 439.4,Z 439.377,A -85,B 0,C 180,E1 -9205.585,E2 -9205.585} C_VEL
LIN {X 0,Y 439.413,Z 439.376,A -85,B 0,C 180,E1 -9208.674,E2 -9208.674} C_VEL
LIN {X 0,Y 439.367,Z 439.384,A -85,B 0,C 180,E1 -9212.031,E2 -9212.031} C_VEL
LIN {X 0,Y 439.392,Z 439.377,A -85,B 0,C 180,E1 -9215.341,E2 -9215.341} C_VEL
LIN {X 0,Y 439.381,Z 439.381,A -85,B 0,C 180,E1 -9218.596,E2 -9218.596} C_VEL
LIN {X 0,Y 439.387,Z 439.377,A -85,B 0,C 180,E1 -9221.258,E2 -9221.258} C_VEL
LIN {X 0,Y 439.404,Z 439.375,A -85,B 0,C 180,E1 -9224.729,E2 -9224.729} C_VEL
LIN {X 0,Y 439.396,Z 439.378,A -85,B 0,C 180,E1 -9227.797,E2 -9227.797} C_VEL
LIN {X 0,Y 439.45,Z 439.371,A -85,B 0,C 180,E1 -9230.231,E2 -9230.231} C_VEL
LIN {X 0,Y 439.377,Z 439.381,A -85,B 0,C 180,E1 -9233.714,E2 -9233.714} C_VEL
LIN {X 0,Y 439.373,Z 439.38,A -85,B 0,C 180,E1 -9237.055,E2 -9237.055} C_VEL
LIN {X 0,Y 439.398,Z 439.378,A -85,B 0,C 180,E1 -9240.276,E2 -9240.276} C_VEL
LIN {X 0,Y 439.435,Z 439.375,A -85,B 0,C 180,E1 -9243.589,E2 -9243.589} C_VEL
LIN {X 0,Y 439.389,Z 439.378,A -85,B 0,C 180,E1 -9246.43,E2 -9246.43} C_VEL
LIN {X 0,Y 439.391,Z 439.38,A -85,B 0,C 180,E1 -9249.398,E2 -9249.398} C_VEL
LIN {X 0,Y 439.434,Z 439.371,A -85,B 0,C 180,E1 -9252.31,E2 -9252.31} C_VEL
LIN {X 0,Y 439.451,Z 439.371,A -85,B 0,C 180,E1 -9255.174,E2 -9255.174} C_VEL
LIN {X 0,Y 439.487,Z 439.366,A -85,B 0,C 180,E1 -9258.002,E2 -9258.002} C_VEL
LIN {X 0,Y 439.537,Z 439.361,A -85,B 0,C 180,E1 -9261.726,E2 -9261.726} C_VEL
LIN {X 0,Y 439.614,Z 439.349,A -85,B 0,C 180,E1 -9264.496,E2 -9264.496} C_VEL
LIN {X 0,Y 439.64,Z 439.347,A -85,B 0,C 180,E1 -9268.168,E2 -9268.168} C_VEL
LIN {X 0,Y 439.767,Z 439.33,A -85,B 0,C 180,E1 -9270,E2 -9270} C_VEL
LIN {X 0,Y 439.613,Z 439.35,A -85,B 0,C 180,E1 -9271,E2 -9271} C_VEL
LIN {X 0,Y 438.905,Z 439.439,A -85,B 0,C 180,E1 -9271.764,E2 -9271.764} C_VEL
LIN {X 0,Y 435.931,Z 439.81,A -85,B 0,C 180,E1 -9273.003,E2 -9273.003} C_VEL
LIN {X 0,Y 433.479,Z 440.114,A -85,B 0,C 180,E1 -9274.004,E2 -9274.004} C_VEL
LIN {X 0,Y 432.506,Z 440.235,A -85,B 0,C 180,E1 -9274.778,E2 -9274.778} C_VEL
LIN {X 0,Y 432.469,Z 440.238,A -85,B 0,C 180,E1 -9275.04,E2 -9275.04} C_VEL
LIN {X 0,Y 432.543,Z 440.233,A -85,B 0,C 180,E1 -9277.632,E2 -9277.632} C_VEL
LIN {X 0,Y 432.397,Z 440.25,A -85,B 0,C 180,E1 -9281.247,E2 -9281.247} C_VEL
LIN {X 0,Y 432.377,Z 440.25,A -85,B 0,C 180,E1 -9284.112,E2 -9284.112} C_VEL
LIN {X 0,Y 432.4,Z 440.25,A -85,B 0,C 180,E1 -9287.011,E2 -9287.011} C_VEL
LIN {X 0,Y 432.341,Z 440.256,A -85,B 0,C 180,E1 -9289.96,E2 -9289.96} C_VEL
LIN {X 0,Y 432.322,Z 440.261,A -85,B 0,C 180,E1 -9292.964,E2 -9292.964} C_VEL
LIN {X 0,Y 432.366,Z 440.252,A -85,B 0,C 180,E1 -9296.032,E2 -9296.032} C_VEL
LIN {X 0,Y 432.344,Z 440.257,A -85,B 0,C 180,E1 -9299.187,E2 -9299.187} C_VEL
LIN {X 0,Y 432.314,Z 440.259,A -85,B 0,C 180,E1 -9302.443,E2 -9302.443} C_VEL
LIN {X 0,Y 432.258,Z 440.269,A -85,B 0,C 180,E1 -9304.684,E2 -9304.684} C_VEL
LIN {X 0,Y 431.975,Z 440.305,A -85,B 0,C 180,E1 -9307.136,E2 -9307.136} C_VEL
LIN {X 0,Y 431.633,Z 440.425,A -85,B 0,C 180,E1 -9310.068,E2 -9310.068} C_VEL
LIN {X 0,Y 431.588,Z 443.19,A -85,B 0,C 180,E1 -9313.151,E2 -9313.151} C_VEL
LIN {X 0,Y 431.533,Z 445.573,A -85,B 0,C 180,E1 -9315.773,E2 -9315.773} C_VEL
LIN {X 0,Y 431.453,Z 448.901,A -85,B 0,C 180,E1 -9319.34,E2 -9319.34} C_VEL
LIN {X 0,Y 431.42,Z 451.421,A -85,B 0,C 180,E1 -9322.008,E2 -9322.008} C_VEL
LIN {X 0,Y 435.922,Z 467.658,A -85,B 0,C 180,E1 -9322.725,E2 -9322.725} C_VEL
LIN {X 0,Y 437.776,Z 475.172,A -85,B 0,C 180,E1 -9323.126,E2 -9323.126} C_VEL
LIN {X 0,Y 437.167,Z 489.249,A -85,B 0,C 180,E1 -9323.857,E2 -9323.857} C_VEL
LIN {X 0,Y 436.397,Z 501.772,A -85,B 0,C 180,E1 -9324.688,E2 -9324.688} C_VEL
LIN {X 0,Y 435.557,Z 514.592,A -85,B 0,C 180,E1 -9325.755,E2 -9325.755} C_VEL
LIN {X 0,Y 434.755,Z 525.441,A -85,B 0,C 180,E1 -9326.858,E2 -9326.858} C_VEL
LIN {X 0,Y 433.94,Z 536.656,A -85,B 0,C 180,E1 -9328.24,E2 -9328.24} C_VEL
LIN {X 0,Y 433.297,Z 545.234,A -85,B 0,C 180,E1 -9329.519,E2 -9329.519} C_VEL
LIN {X 0,Y 432.694,Z 552.695,A -85,B 0,C 180,E1 -9330.838,E2 -9330.838} C_VEL
LIN {X 0,Y 432.233,Z 559.995,A -85,B 0,C 180,E1 -9332.393,E2 -9332.393} C_VEL
LIN {X 0,Y 431.891,Z 565.883,A -85,B 0,C 180,E1 -9333.937,E2 -9333.937} C_VEL
LIN {X 0,Y 431.552,Z 571.399,A -85,B 0,C 180,E1 -9335.778,E2 -9335.778} C_VEL
LIN {X 0,Y 431.394,Z 574.162,A -85,B 0,C 180,E1 -9336.983,E2 -9336.983} C_VEL
LIN {X 0,Y 431.299,Z 576.408,A -85,B 0,C 180,E1 -9338.248,E2 -9338.248} C_VEL
LIN {X 0,Y 431.183,Z 578.461,A -85,B 0,C 180,E1 -9339.983,E2 -9339.983} C_VEL
LIN {X 0,Y 431.209,Z 579.116,A -85,B 0,C 180,E1 -9340.976,E2 -9340.976} C_VEL
LIN {X 0,Y 431.145,Z 579.316,A -85,B 0,C 180,E1 -9342.937,E2 -9342.937} C_VEL
LIN {X 0,Y 431.245,Z 578.017,A -85,B 0,C 180,E1 -9344.885,E2 -9344.885} C_VEL
LIN {X 0,Y 431.394,Z 575.271,A -85,B 0,C 180,E1 -9346.816,E2 -9346.816} C_VEL
LIN {X 0,Y 431.686,Z 571.035,A -85,B 0,C 180,E1 -9348.734,E2 -9348.734} C_VEL
LIN {X 0,Y 432.069,Z 565.224,A -85,B 0,C 180,E1 -9350.638,E2 -9350.638} C_VEL
LIN {X 0,Y 432.554,Z 558.457,A -85,B 0,C 180,E1 -9352.346,E2 -9352.346} C_VEL
LIN {X 0,Y 433.21,Z 550.516,A -85,B 0,C 180,E1 -9353.947,E2 -9353.947} C_VEL
LIN {X 0,Y 433.853,Z 542.052,A -85,B 0,C 180,E1 -9355.354,E2 -9355.354} C_VEL
LIN {X 0,Y 434.71,Z 531.811,A -85,B 0,C 180,E1 -9356.756,E2 -9356.756} C_VEL
LIN {X 0,Y 435.615,Z 520.438,A -85,B 0,C 180,E1 -9358.035,E2 -9358.035} C_VEL
LIN {X 0,Y 436.57,Z 507.78,A -85,B 0,C 180,E1 -9359.193,E2 -9359.193} C_VEL
LIN {X 0,Y 437.455,Z 494.613,A -85,B 0,C 180,E1 -9360.157,E2 -9360.157} C_VEL
LIN {X 0,Y 438.254,Z 481.233,A -85,B 0,C 180,E1 -9360.919,E2 -9360.919} C_VEL
LIN {X 0,Y 438.216,Z 475.231,A -85,B 0,C 180,E1 -9361.218,E2 -9361.218} C_VEL
LIN {X 0,Y 434.361,Z 461.994,A -85,B 0,C 180,E1 -9361.956,E2 -9361.956} C_VEL
LIN {X 0,Y 431.712,Z 454.141,A -85,B 0,C 180,E1 -9362.361,E2 -9362.361} C_VEL
LIN {X 0,Y 432.05,Z 452.303,A -85,B 0,C 180,E1 -9364.665,E2 -9364.665} C_VEL
LIN {X 0,Y 432.126,Z 450.186,A -85,B 0,C 180,E1 -9367.476,E2 -9367.476} C_VEL
LIN {X 0,Y 432.106,Z 448.157,A -85,B 0,C 180,E1 -9370.306,E2 -9370.306} C_VEL
LIN {X 0,Y 432.225,Z 446.195,A -85,B 0,C 180,E1 -9373.158,E2 -9373.158} C_VEL
LIN {X 0,Y 432.387,Z 444.068,A -85,B 0,C 180,E1 -9376.47,E2 -9376.47} C_VEL
LIN {X 0,Y 432.521,Z 442.273,A -85,B 0,C 180,E1 -9379.538,E2 -9379.538} C_VEL
LIN {X 0,Y 432.436,Z 440.973,A -85,B 0,C 180,E1 -9382.127,E2 -9382.127} C_VEL
LIN {X 0,Y 432.378,Z 440.254,A -85,B 0,C 180,E1 -9384.464,E2 -9384.464} C_VEL
LIN {X 0,Y 432.387,Z 440.252,A -85,B 0,C 180,E1 -9387.072,E2 -9387.072} C_VEL
LIN {X 0,Y 432.363,Z 440.254,A -85,B 0,C 180,E1 -9390.515,E2 -9390.515} C_VEL
LIN {X 0,Y 432.355,Z 440.256,A -85,B 0,C 180,E1 -9394.004,E2 -9394.004} C_VEL
LIN {X 0,Y 432.329,Z 440.26,A -85,B 0,C 180,E1 -9397.199,E2 -9397.199} C_VEL
LIN {X 0,Y 432.356,Z 440.336,A -85,B 0,C 180,E1 -9398.718,E2 -9398.718} C_VEL
LIN {X 0,Y 432.734,Z 442.411,A -85,B 0,C 180,E1 -9401.75,E2 -9401.75} C_VEL
LIN {X 0,Y 433.186,Z 445.019,A -85,B 0,C 180,E1 -9404.452,E2 -9404.452} C_VEL
LIN {X 0,Y 433.726,Z 448.2,A -85,B 0,C 180,E1 -9407.114,E2 -9407.114} C_VEL
LIN {X 0,Y 434.333,Z 451.781,A -85,B 0,C 180,E1 -9409.667,E2 -9409.667} C_VEL
LIN {X 0,Y 434.492,Z 453.798,A -85,B 0,C 180,E1 -9410.933,E2 -9410.933} C_VEL
LIN {X 0,Y 434.375,Z 456.431,A -85,B 0,C 180,E1 -9412.448,E2 -9412.448} C_VEL
LIN {X 0,Y 433.672,Z 462.765,A -85,B 0,C 180,E1 -9415.74,E2 -9415.74} C_VEL
LIN {X 0,Y 433.158,Z 469.062,A -85,B 0,C 180,E1 -9418.722,E2 -9418.722} C_VEL
LIN {X 0,Y 432.784,Z 474.776,A -85,B 0,C 180,E1 -9421.272,E2 -9421.272} C_VEL
LIN {X 0,Y 432.329,Z 482.364,A -85,B 0,C 180,E1 -9424.483,E2 -9424.483} C_VEL
LIN {X 0,Y 431.996,Z 491.159,A -85,B 0,C 180,E1 -9428.027,E2 -9428.027} C_VEL
LIN {X 0,Y 431.84,Z 495.453,A -85,B 0,C 180,E1 -9429.628,E2 -9429.628} C_VEL
LIN {X 0,Y 434.947,Z 510.607,A -85,B 0,C 180,E1 -9430.232,E2 -9430.232} C_VEL
LIN {X 0,Y 436.876,Z 525.05,A -85,B 0,C 180,E1 -9430.939,E2 -9430.939} C_VEL
LIN {X 0,Y 437.307,Z 529.446,A -85,B 0,C 180,E1 -9431.178,E2 -9431.178} C_VEL
LIN {X 0,Y 436.476,Z 542.948,A -85,B 0,C 180,E1 -9431.957,E2 -9431.957} C_VEL
LIN {X 0,Y 435.565,Z 555.578,A -85,B 0,C 180,E1 -9432.875,E2 -9432.875} C_VEL
LIN {X 0,Y 434.522,Z 568.559,A -85,B 0,C 180,E1 -9434.041,E2 -9434.041} C_VEL
LIN {X 0,Y 433.707,Z 579.267,A -85,B 0,C 180,E1 -9435.214,E2 -9435.214} C_VEL
LIN {X 0,Y 432.976,Z 589.974,A -85,B 0,C 180,E1 -9436.626,E2 -9436.626} C_VEL
LIN {X 0,Y 432.394,Z 598.857,A -85,B 0,C 180,E1 -9438.04,E2 -9438.04} C_VEL
LIN {X 0,Y 431.869,Z 607.43,A -85,B 0,C 180,E1 -9439.688,E2 -9439.688} C_VEL
LIN {X 0,Y 431.58,Z 613.426,A -85,B 0,C 180,E1 -9441.101,E2 -9441.101} C_VEL
LIN {X 0,Y 431.394,Z 618.364,A -85,B 0,C 180,E1 -9442.511,E2 -9442.511} C_VEL
LIN {X 0,Y 431.399,Z 621.54,A -85,B 0,C 180,E1 -9443.597,E2 -9443.597} C_VEL
LIN {X 0,Y 431.265,Z 625.474,A -85,B 0,C 180,E1 -9445.326,E2 -9445.326} C_VEL
LIN {X 0,Y 431.31,Z 628.334,A -85,B 0,C 180,E1 -9447.198,E2 -9447.198} C_VEL
LIN {X 0,Y 431.274,Z 629.766,A -85,B 0,C 180,E1 -9449.066,E2 -9449.066} C_VEL
LIN {X 0,Y 431.287,Z 629.801,A -85,B 0,C 180,E1 -9450.934,E2 -9450.934} C_VEL
LIN {X 0,Y 431.304,Z 628.447,A -85,B 0,C 180,E1 -9452.802,E2 -9452.802} C_VEL
LIN {X 0,Y 431.259,Z 625.675,A -85,B 0,C 180,E1 -9454.674,E2 -9454.674} C_VEL
LIN {X 0,Y 431.372,Z 621.418,A -85,B 0,C 180,E1 -9456.548,E2 -9456.548} C_VEL
LIN {X 0,Y 431.505,Z 615.545,A -85,B 0,C 180,E1 -9458.429,E2 -9458.429} C_VEL
LIN {X 0,Y 431.811,Z 608.917,A -85,B 0,C 180,E1 -9460.076,E2 -9460.076} C_VEL
LIN {X 0,Y 432.334,Z 600.686,A -85,B 0,C 180,E1 -9461.724,E2 -9461.724} C_VEL
LIN {X 0,Y 432.875,Z 592.067,A -85,B 0,C 180,E1 -9463.138,E2 -9463.138} C_VEL
LIN {X 0,Y 433.642,Z 581.647,A -85,B 0,C 180,E1 -9464.549,E2 -9464.549} C_VEL
LIN {X 0,Y 434.467,Z 570.031,A -85,B 0,C 180,E1 -9465.841,E2 -9465.841} C_VEL
LIN {X 0,Y 435.483,Z 557.095,A -85,B 0,C 180,E1 -9467.008,E2 -9467.008} C_VEL
LIN {X 0,Y 436.371,Z 544.083,A -85,B 0,C 180,E1 -9467.949,E2 -9467.949} C_VEL
LIN {X 0,Y 437.216,Z 529.713,A -85,B 0,C 180,E1 -9468.753,E2 -9468.753} C_VEL
LIN {X 0,Y 435.498,Z 516.949,A -85,B 0,C 180,E1 -9469.383,E2 -9469.383} C_VEL
LIN {X 0,Y 432.785,Z 502.193,A -85,B 0,C 180,E1 -9469.954,E2 -9469.954} C_VEL
LIN {X 0,Y 431.958,Z 497.667,A -85,B 0,C 180,E1 -9470.102,E2 -9470.102} C_VEL
LIN {X 0,Y 432.272,Z 489.231,A -85,B 0,C 180,E1 -9473.473,E2 -9473.473} C_VEL
LIN {X 0,Y 432.705,Z 481.295,A -85,B 0,C 180,E1 -9476.708,E2 -9476.708} C_VEL
LIN {X 0,Y 433.154,Z 473.009,A -85,B 0,C 180,E1 -9480.197,E2 -9480.197} C_VEL
LIN {X 0,Y 433.69,Z 465.547,A -85,B 0,C 180,E1 -9483.433,E2 -9483.433} C_VEL
LIN {X 0,Y 434.236,Z 458.107,A -85,B 0,C 180,E1 -9486.786,E2 -9486.786} C_VEL
LIN {X 0,Y 434.447,Z 453.146,A -85,B 0,C 180,E1 -9489.116,E2 -9489.116} C_VEL
LIN {X 0,Y 434.015,Z 449.382,A -85,B 0,C 180,E1 -9490.993,E2 -9490.993} C_VEL
LIN {X 0,Y 432.858,Z 442.931,A -85,B 0,C 180,E1 -9494.406,E2 -9494.406} C_VEL
LIN {X 0,Y 432.378,Z 440.252,A -85,B 0,C 180,E1 -9495.983,E2 -9495.983} C_VEL
LIN {X 0,Y 432.364,Z 440.252,A -85,B 0,C 180,E1 -9498.392,E2 -9498.392} C_VEL
LIN {X 0,Y 432.335,Z 440.26,A -85,B 0,C 180,E1 -9501.85,E2 -9501.85} C_VEL
LIN {X 0,Y 432.336,Z 440.258,A -85,B 0,C 180,E1 -9505.323,E2 -9505.323} C_VEL
LIN {X 0,Y 432.329,Z 440.258,A -85,B 0,C 180,E1 -9508.655,E2 -9508.655} C_VEL
LIN {X 0,Y 432.379,Z 440.25,A -85,B 0,C 180,E1 -9511.877,E2 -9511.877} C_VEL
LIN {X 0,Y 432.346,Z 440.257,A -85,B 0,C 180,E1 -9514.999,E2 -9514.999} C_VEL
LIN {X 0,Y 432.352,Z 440.253,A -85,B 0,C 180,E1 -9518.046,E2 -9518.046} C_VEL
LIN {X 0,Y 432.38,Z 440.254,A -85,B 0,C 180,E1 -9521.029,E2 -9521.029} C_VEL
LIN {X 0,Y 432.424,Z 440.245,A -85,B 0,C 180,E1 -9523.961,E2 -9523.961} C_VEL
LIN {X 0,Y 432.453,Z 440.241,A -85,B 0,C 180,E1 -9527.803,E2 -9527.803} C_VEL
LIN {X 0,Y 432.486,Z 440.237,A -85,B 0,C 180,E1 -9531.59,E2 -9531.59} C_VEL
LIN {X 0,Y 432.592,Z 440.225,A -85,B 0,C 180,E1 -9534.406,E2 -9534.406} C_VEL
LIN {X 0,Y 432.6,Z 440.225,A -85,B 0,C 180,E1 -9538.138,E2 -9538.138} C_VEL
LIN {X 0,Y 432.727,Z 440.207,A -85,B 0,C 180,E1 -9540,E2 -9540} C_VEL
LIN {X 0,Y 432.601,Z 440.226,A -85,B 0,C 180,E1 -9542.794,E2 -9542.794} C_VEL
LIN {X 0,Y 432.571,Z 440.229,A -85,B 0,C 180,E1 -9546.531,E2 -9546.531} C_VEL
LIN {X 0,Y 432.437,Z 440.243,A -85,B 0,C 180,E1 -9549.353,E2 -9549.353} C_VEL
LIN {X 0,Y 432.425,Z 440.246,A -85,B 0,C 180,E1 -9552.804,E2 -9552.804} C_VEL
LIN {X 0,Y 432.407,Z 440.25,A -85,B 0,C 180,E1 -9556.479,E2 -9556.479} C_VEL
LIN {X 0,Y 432.334,Z 440.259,A -85,B 0,C 180,E1 -9559.961,E2 -9559.961} C_VEL
LIN {X 0,Y 432.315,Z 440.259,A -85,B 0,C 180,E1 -9562.965,E2 -9562.965} C_VEL
LIN {X 0,Y 432.359,Z 440.255,A -85,B 0,C 180,E1 -9566.033,E2 -9566.033} C_VEL
LIN {X 0,Y 432.339,Z 440.256,A -85,B 0,C 180,E1 -9569.188,E2 -9569.188} C_VEL
LIN {X 0,Y 432.319,Z 440.259,A -85,B 0,C 180,E1 -9572.444,E2 -9572.444} C_VEL
LIN {X 0,Y 432.342,Z 440.256,A -85,B 0,C 180,E1 -9575.633,E2 -9575.633} C_VEL
LIN {X 0,Y 432.344,Z 440.256,A -85,B 0,C 180,E1 -9578.716,E2 -9578.716} C_VEL
LIN {X 0,Y 432.333,Z 440.26,A -85,B 0,C 180,E1 -9581.798,E2 -9581.798} C_VEL
LIN {X 0,Y 432.339,Z 440.257,A -85,B 0,C 180,E1 -9584.347,E2 -9584.347} C_VEL
LIN {X 0,Y 432.319,Z 440.258,A -85,B 0,C 180,E1 -9587.016,E2 -9587.016} C_VEL
LIN {X 0,Y 432.355,Z 440.257,A -85,B 0,C 180,E1 -9589.818,E2 -9589.818} C_VEL
LIN {X 0,Y 432.317,Z 440.258,A -85,B 0,C 180,E1 -9593.024,E2 -9593.024} C_VEL
LIN {X 0,Y 432.36,Z 440.255,A -85,B 0,C 180,E1 -9595.997,E2 -9595.997} C_VEL
LIN {X 0,Y 432.396,Z 440.251,A -85,B 0,C 180,E1 -9599.745,E2 -9599.745} C_VEL
LIN {X 0,Y 432.402,Z 440.249,A -85,B 0,C 180,E1 -9603.373,E2 -9603.373} C_VEL
LIN {X 0,Y 432.373,Z 440.254,A -85,B 0,C 180,E1 -9606.024,E2 -9606.024} C_VEL
LIN {X 0,Y 432.353,Z 440.255,A -85,B 0,C 180,E1 -9609.047,E2 -9609.047} C_VEL
LIN {X 0,Y 432.381,Z 440.251,A -85,B 0,C 180,E1 -9612.012,E2 -9612.012} C_VEL
LIN {X 0,Y 432.399,Z 440.249,A -85,B 0,C 180,E1 -9614.927,E2 -9614.927} C_VEL
LIN {X 0,Y 432.463,Z 440.242,A -85,B 0,C 180,E1 -9617.804,E2 -9617.804} C_VEL
LIN {X 0,Y 432.486,Z 440.24,A -85,B 0,C 180,E1 -9621.59,E2 -9621.59} C_VEL
LIN {X 0,Y 432.59,Z 440.224,A -85,B 0,C 180,E1 -9624.406,E2 -9624.406} C_VEL
LIN {X 0,Y 432.61,Z 440.223,A -85,B 0,C 180,E1 -9628.138,E2 -9628.138} C_VEL
LIN {X 0,Y 432.736,Z 440.206,A -85,B 0,C 180,E1 -9630,E2 -9630} C_VEL
LIN {X 0,Y 432.596,Z 440.225,A -85,B 0,C 180,E1 -9632.794,E2 -9632.794} C_VEL
LIN {X 0,Y 432.469,Z 440.238,A -85,B 0,C 180,E1 -9635.04,E2 -9635.04} C_VEL
LIN {X 0,Y 431.91,Z 440.31,A -85,B 0,C 180,E1 -9635.819,E2 -9635.819} C_VEL
LIN {X 0,Y 429.059,Z 440.666,A -85,B 0,C 180,E1 -9637.083,E2 -9637.083} C_VEL
LIN {X 0,Y 426.572,Z 440.974,A -85,B 0,C 180,E1 -9638.103,E2 -9638.103} C_VEL
LIN {X 0,Y 425.492,Z 441.109,A -85,B 0,C 180,E1 -9638.893,E2 -9638.893} C_VEL
LIN {X 0,Y 425.403,Z 441.119,A -85,B 0,C 180,E1 -9639.16,E2 -9639.16} C_VEL
LIN {X 0,Y 425.397,Z 441.122,A -85,B 0,C 180,E1 -9642.903,E2 -9642.903} C_VEL
LIN {X 0,Y 425.365,Z 441.126,A -85,B 0,C 180,E1 -9646.605,E2 -9646.605} C_VEL
LIN {X 0,Y 425.331,Z 441.13,A -85,B 0,C 180,E1 -9649.635,E2 -9649.635} C_VEL
LIN {X 0,Y 425.309,Z 441.133,A -85,B 0,C 180,E1 -9653.365,E2 -9653.365} C_VEL
LIN {X 0,Y 425.35,Z 441.128,A -85,B 0,C 180,E1 -9656.844,E2 -9656.844} C_VEL
LIN {X 0,Y 425.292,Z 441.134,A -85,B 0,C 180,E1 -9659.719,E2 -9659.719} C_VEL
LIN {X 0,Y 425.26,Z 441.139,A -85,B 0,C 180,E1 -9663.049,E2 -9663.049} C_VEL
LIN {X 0,Y 425.087,Z 441.16,A -85,B 0,C 180,E1 -9665.892,E2 -9665.892} C_VEL
LIN {X 0,Y 424.725,Z 441.209,A -85,B 0,C 180,E1 -9668.96,E2 -9668.96} C_VEL
LIN {X 0,Y 424.551,Z 441.438,A -85,B 0,C 180,E1 -9670.404,E2 -9670.404} C_VEL
LIN {X 0,Y 424.519,Z 443.966,A -85,B 0,C 180,E1 -9673.245,E2 -9673.245} C_VEL
LIN {X 0,Y 424.438,Z 447.166,A -85,B 0,C 180,E1 -9676.765,E2 -9676.765} C_VEL
LIN {X 0,Y 424.36,Z 449.952,A -85,B 0,C 180,E1 -9679.767,E2 -9679.767} C_VEL
LIN {X 0,Y 424.337,Z 451.788,A -85,B 0,C 180,E1 -9681.71,E2 -9681.71} C_VEL
LIN {X 0,Y 428.59,Z 466.959,A -85,B 0,C 180,E1 -9682.373,E2 -9682.373} C_VEL
LIN {X 0,Y 430.998,Z 476.463,A -85,B 0,C 180,E1 -9682.891,E2 -9682.891} C_VEL
LIN {X 0,Y 430.339,Z 490.638,A -85,B 0,C 180,E1 -9683.652,E2 -9683.652} C_VEL
LIN {X 0,Y 429.55,Z 502.883,A -85,B 0,C 180,E1 -9684.491,E2 -9684.491} C_VEL
LIN {X 0,Y 428.683,Z 515.367,A -85,B 0,C 180,E1 -9685.555,E2 -9685.555} C_VEL
LIN {X 0,Y 427.728,Z 527.509,A -85,B 0,C 180,E1 -9686.827,E2 -9686.827} C_VEL
LIN {X 0,Y 426.902,Z 538.215,A -85,B 0,C 180,E1 -9688.21,E2 -9688.21} C_VEL
LIN {X 0,Y 426.205,Z 546.773,A -85,B 0,C 180,E1 -9689.532,E2 -9689.532} C_VEL
LIN {X 0,Y 425.596,Z 555.016,A -85,B 0,C 180,E1 -9691.067,E2 -9691.067} C_VEL
LIN {X 0,Y 425.18,Z 561.111,A -85,B 0,C 180,E1 -9692.43,E2 -9692.43} C_VEL
LIN {X 0,Y 424.8,Z 566.859,A -85,B 0,C 180,E1 -9693.996,E2 -9693.996} C_VEL
LIN {X 0,Y 424.511,Z 571.484,A -85,B 0,C 180,E1 -9695.58,E2 -9695.58} C_VEL
LIN {X 0,Y 424.303,Z 574.893,A -85,B 0,C 180,E1 -9697.092,E2 -9697.092} C_VEL
LIN {X 0,Y 424.187,Z 577.423,A -85,B 0,C 180,E1 -9698.623,E2 -9698.623} C_VEL
LIN {X 0,Y 424.1,Z 579.352,A -85,B 0,C 180,E1 -9700.644,E2 -9700.644} C_VEL
LIN {X 0,Y 424.098,Z 579.75,A -85,B 0,C 180,E1 -9701.647,E2 -9701.647} C_VEL
LIN {X 0,Y 424.098,Z 579.446,A -85,B 0,C 180,E1 -9703.637,E2 -9703.637} C_VEL
LIN {X 0,Y 424.2,Z 577.701,A -85,B 0,C 180,E1 -9705.61,E2 -9705.61} C_VEL
LIN {X 0,Y 424.43,Z 574.485,A -85,B 0,C 180,E1 -9707.569,E2 -9707.569} C_VEL
LIN {X 0,Y 424.667,Z 571.067,A -85,B 0,C 180,E1 -9709.028,E2 -9709.028} C_VEL
LIN {X 0,Y 424.983,Z 566.739,A -85,B 0,C 180,E1 -9710.481,E2 -9710.481} C_VEL
LIN {X 0,Y 425.5,Z 559.869,A -85,B 0,C 180,E1 -9712.309,E2 -9712.309} C_VEL
LIN {X 0,Y 426.179,Z 552.626,A -85,B 0,C 180,E1 -9713.846,E2 -9713.846} C_VEL
LIN {X 0,Y 426.831,Z 544.488,A -85,B 0,C 180,E1 -9715.277,E2 -9715.277} C_VEL
LIN {X 0,Y 427.676,Z 534.717,A -85,B 0,C 180,E1 -9716.703,E2 -9716.703} C_VEL
LIN {X 0,Y 428.641,Z 523.918,A -85,B 0,C 180,E1 -9718.003,E2 -9718.003} C_VEL
LIN {X 0,Y 429.58,Z 511.97,A -85,B 0,C 180,E1 -9719.18,E2 -9719.18} C_VEL
LIN {X 0,Y 430.57,Z 498.643,A -85,B 0,C 180,E1 -9720.234,E2 -9720.234} C_VEL
LIN {X 0,Y 431.397,Z 486.006,A -85,B 0,C 180,E1 -9721.025,E2 -9721.025} C_VEL
LIN {X 0,Y 431.758,Z 477.856,A -85,B 0,C 180,E1 -9721.449,E2 -9721.449} C_VEL
LIN {X 0,Y 428.445,Z 465.775,A -85,B 0,C 180,E1 -9722.163,E2 -9722.163} C_VEL
LIN {X 0,Y 424.699,Z 454.711,A -85,B 0,C 180,E1 -9722.756,E2 -9722.756} C_VEL
LIN {X 0,Y 425.02,Z 453.158,A -85,B 0,C 180,E1 -9724.742,E2 -9724.742} C_VEL
LIN {X 0,Y 425.096,Z 451.04,A -85,B 0,C 180,E1 -9727.6,E2 -9727.6} C_VEL
LIN {X 0,Y 425.124,Z 448.374,A -85,B 0,C 180,E1 -9731.442,E2 -9731.442} C_VEL
LIN {X 0,Y 425.21,Z 447.101,A -85,B 0,C 180,E1 -9733.379,E2 -9733.379} C_VEL
LIN {X 0,Y 425.401,Z 445.061,A -85,B 0,C 180,E1 -9736.626,E2 -9736.626} C_VEL
LIN {X 0,Y 425.53,Z 443.346,A -85,B 0,C 180,E1 -9739.714,E2 -9739.714} C_VEL
LIN {X 0,Y 425.42,Z 442.119,A -85,B 0,C 180,E1 -9742.331,E2 -9742.331} C_VEL
LIN {X 0,Y 425.325,Z 441.199,A -85,B 0,C 180,E1 -9744.661,E2 -9744.661} C_VEL
LIN {X 0,Y 425.345,Z 441.129,A -85,B 0,C 180,E1 -9747.558,E2 -9747.558} C_VEL
LIN {X 0,Y 425.292,Z 441.135,A -85,B 0,C 180,E1 -9750.816,E2 -9750.816} C_VEL
LIN {X 0,Y 425.307,Z 441.135,A -85,B 0,C 180,E1 -9754.288,E2 -9754.288} C_VEL
LIN {X 0,Y 425.336,Z 441.367,A -85,B 0,C 180,E1 -9757.688,E2 -9757.688} C_VEL
LIN {X 0,Y 425.687,Z 443.083,A -85,B 0,C 180,E1 -9760.586,E2 -9760.586} C_VEL
LIN {X 0,Y 426.144,Z 445.909,A -85,B 0,C 180,E1 -9763.842,E2 -9763.842} C_VEL
LIN {X 0,Y 426.646,Z 448.821,A -85,B 0,C 180,E1 -9766.452,E2 -9766.452} C_VEL
LIN {X 0,Y 427.273,Z 452.442,A -85,B 0,C 180,E1 -9769.168,E2 -9769.168} C_VEL
LIN {X 0,Y 427.478,Z 455.84,A -85,B 0,C 180,E1 -9771.338,E2 -9771.338} C_VEL
LIN {X 0,Y 427.214,Z 458.92,A -85,B 0,C 180,E1 -9773.098,E2 -9773.098} C_VEL
LIN {X 0,Y 426.545,Z 465.469,A -85,B 0,C 180,E1 -9776.499,E2 -9776.499} C_VEL
LIN {X 0,Y 425.971,Z 472.421,A -85,B 0,C 180,E1 -9779.788,E2 -9779.788} C_VEL
LIN {X 0,Y 425.454,Z 479.939,A -85,B 0,C 180,E1 -9783.128,E2 -9783.128} C_VEL
LIN {X 0,Y 425.019,Z 488.271,A -85,B 0,C 180,E1 -9786.619,E2 -9786.619} C_VEL
LIN {X 0,Y 424.785,Z 494.649,A -85,B 0,C 180,E1 -9789.193,E2 -9789.193} C_VEL
LIN {X 0,Y 428.339,Z 512.016,A -85,B 0,C 180,E1 -9789.947,E2 -9789.947} C_VEL
LIN {X 0,Y 430.26,Z 527.056,A -85,B 0,C 180,E1 -9790.724,E2 -9790.724} C_VEL
LIN {X 0,Y 430.483,Z 530.847,A -85,B 0,C 180,E1 -9790.943,E2 -9790.943} C_VEL
LIN {X 0,Y 429.498,Z 544.948,A -85,B 0,C 180,E1 -9791.806,E2 -9791.806} C_VEL
LIN {X 0,Y 428.534,Z 558.149,A -85,B 0,C 180,E1 -9792.831,E2 -9792.831} C_VEL
LIN {X 0,Y 427.491,Z 570.576,A -85,B 0,C 180,E1 -9794.016,E2 -9794.016} C_VEL
LIN {X 0,Y 426.647,Z 580.89,A -85,B 0,C 180,E1 -9795.207,E2 -9795.207} C_VEL
LIN {X 0,Y 425.881,Z 591.207,A -85,B 0,C 180,E1 -9796.642,E2 -9796.642} C_VEL
LIN {X 0,Y 425.285,Z 599.818,A -85,B 0,C 180,E1 -9798.079,E2 -9798.079} C_VEL
LIN {X 0,Y 424.763,Z 608.078,A -85,B 0,C 180,E1 -9799.755,E2 -9799.755} C_VEL
LIN {X 0,Y 424.439,Z 614.76,A -85,B 0,C 180,E1 -9801.43,E2 -9801.43} C_VEL
LIN {X 0,Y 424.311,Z 620.72,A -85,B 0,C 180,E1 -9803.342,E2 -9803.342} C_VEL
LIN {X 0,Y 424.193,Z 625.063,A -85,B 0,C 180,E1 -9805.248,E2 -9805.248} C_VEL
LIN {X 0,Y 424.239,Z 627.924,A -85,B 0,C 180,E1 -9807.151,E2 -9807.151} C_VEL
LIN {X 0,Y 424.187,Z 629.348,A -85,B 0,C 180,E1 -9809.051,E2 -9809.051} C_VEL
LIN {X 0,Y 424.2,Z 629.374,A -85,B 0,C 180,E1 -9810.949,E2 -9810.949} C_VEL
LIN {X 0,Y 424.232,Z 628.01,A -85,B 0,C 180,E1 -9812.849,E2 -9812.849} C_VEL
LIN {X 0,Y 424.187,Z 625.222,A -85,B 0,C 180,E1 -9814.752,E2 -9814.752} C_VEL
LIN {X 0,Y 424.294,Z 620.946,A -85,B 0,C 180,E1 -9816.658,E2 -9816.658} C_VEL
LIN {X 0,Y 424.44,Z 615.051,A -85,B 0,C 180,E1 -9818.57,E2 -9818.57} C_VEL
LIN {X 0,Y 424.769,Z 608.398,A -85,B 0,C 180,E1 -9820.245,E2 -9820.245} C_VEL
LIN {X 0,Y 425.293,Z 600.127,A -85,B 0,C 180,E1 -9821.921,E2 -9821.921} C_VEL
LIN {X 0,Y 425.908,Z 591.477,A -85,B 0,C 180,E1 -9823.357,E2 -9823.357} C_VEL
LIN {X 0,Y 426.706,Z 581.013,A -85,B 0,C 180,E1 -9824.791,E2 -9824.791} C_VEL
LIN {X 0,Y 427.589,Z 569.356,A -85,B 0,C 180,E1 -9826.103,E2 -9826.103} C_VEL
LIN {X 0,Y 428.539,Z 557.785,A -85,B 0,C 180,E1 -9827.169,E2 -9827.169} C_VEL
LIN {X 0,Y 429.432,Z 545.17,A -85,B 0,C 180,E1 -9828.116,E2 -9828.116} C_VEL
LIN {X 0,Y 430.351,Z 530.808,A -85,B 0,C 180,E1 -9828.961,E2 -9828.961} C_VEL
LIN {X 0,Y 428.847,Z 518.871,A -85,B 0,C 180,E1 -9829.579,E2 -9829.579} C_VEL
LIN {X 0,Y 426.135,Z 503.785,A -85,B 0,C 180,E1 -9830.209,E2 -9830.209} C_VEL
LIN {X 0,Y 424.895,Z 497.297,A -85,B 0,C 180,E1 -9830.434,E2 -9830.434} C_VEL
LIN {X 0,Y 425.244,Z 488.839,A -85,B 0,C 180,E1 -9833.885,E2 -9833.885} C_VEL
LIN {X 0,Y 425.665,Z 481.561,A -85,B 0,C 180,E1 -9836.928,E2 -9836.928} C_VEL
LIN {X 0,Y 426.131,Z 473.911,A -85,B 0,C 180,E1 -9840.2,E2 -9840.2} C_VEL
LIN {X 0,Y 426.679,Z 466.48,A -85,B 0,C 180,E1 -9843.489,E2 -9843.489} C_VEL
LIN {X 0,Y 427.238,Z 459.037,A -85,B 0,C 180,E1 -9846.899,E2 -9846.899} C_VEL
LIN {X 0,Y 427.493,Z 455.338,A -85,B 0,C 180,E1 -9848.661,E2 -9848.661} C_VEL
LIN {X 0,Y 427.125,Z 451.033,A -85,B 0,C 180,E1 -9850.809,E2 -9850.809} C_VEL
LIN {X 0,Y 425.801,Z 443.643,A -85,B 0,C 180,E1 -9854.787,E2 -9854.787} C_VEL
LIN {X 0,Y 425.318,Z 441.131,A -85,B 0,C 180,E1 -9856.219,E2 -9856.219} C_VEL
LIN {X 0,Y 425.298,Z 441.132,A -85,B 0,C 180,E1 -9858.624,E2 -9858.624} C_VEL
LIN {X 0,Y 425.308,Z 441.133,A -85,B 0,C 180,E1 -9861.102,E2 -9861.102} C_VEL
LIN {X 0,Y 425.295,Z 441.135,A -85,B 0,C 180,E1 -9864.664,E2 -9864.664} C_VEL
LIN {X 0,Y 425.269,Z 441.135,A -85,B 0,C 180,E1 -9868.074,E2 -9868.074} C_VEL
LIN {X 0,Y 425.332,Z 441.13,A -85,B 0,C 180,E1 -9871.368,E2 -9871.368} C_VEL
LIN {X 0,Y 425.29,Z 441.136,A -85,B 0,C 180,E1 -9874.554,E2 -9874.554} C_VEL
LIN {X 0,Y 425.282,Z 441.134,A -85,B 0,C 180,E1 -9877.661,E2 -9877.661} C_VEL
LIN {X 0,Y 425.356,Z 441.127,A -85,B 0,C 180,E1 -9880.704,E2 -9880.704} C_VEL
LIN {X 0,Y 425.382,Z 441.122,A -85,B 0,C 180,E1 -9883.688,E2 -9883.688} C_VEL
LIN {X 0,Y 425.406,Z 441.119,A -85,B 0,C 180,E1 -9887.598,E2 -9887.598} C_VEL
LIN {X 0,Y 425.436,Z 441.115,A -85,B 0,C 180,E1 -9891.45,E2 -9891.45} C_VEL
LIN {X 0,Y 425.548,Z 441.103,A -85,B 0,C 180,E1 -9894.313,E2 -9894.313} C_VEL
LIN {X 0,Y 425.57,Z 441.101,A -85,B 0,C 180,E1 -9898.107,E2 -9898.107} C_VEL
LIN {X 0,Y 425.696,Z 441.083,A -85,B 0,C 180,E1 -9900,E2 -9900} C_VEL
LIN {X 0,Y 425.553,Z 441.104,A -85,B 0,C 180,E1 -9902.84,E2 -9902.84} C_VEL
LIN {X 0,Y 425.573,Z 441.098,A -85,B 0,C 180,E1 -9905.687,E2 -9905.687} C_VEL
LIN {X 0,Y 425.436,Z 441.119,A -85,B 0,C 180,E1 -9908.55,E2 -9908.55} C_VEL
LIN {X 0,Y 425.406,Z 441.122,A -85,B 0,C 180,E1 -9912.402,E2 -9912.402} C_VEL
LIN {X 0,Y 425.383,Z 441.124,A -85,B 0,C 180,E1 -9916.312,E2 -9916.312} C_VEL
LIN {X 0,Y 425.323,Z 441.13,A -85,B 0,C 180,E1 -9919.636,E2 -9919.636} C_VEL
LIN {X 0,Y 425.302,Z 441.131,A -85,B 0,C 180,E1 -9923.366,E2 -9923.366} C_VEL
LIN {X 0,Y 425.342,Z 441.127,A -85,B 0,C 180,E1 -9926.845,E2 -9926.845} C_VEL
LIN {X 0,Y 425.287,Z 441.136,A -85,B 0,C 180,E1 -9929.72,E2 -9929.72} C_VEL
LIN {X 0,Y 425.279,Z 441.135,A -85,B 0,C 180,E1 -9933.049,E2 -9933.049} C_VEL
LIN {X 0,Y 425.281,Z 441.137,A -85,B 0,C 180,E1 -9935.93,E2 -9935.93} C_VEL
LIN {X 0,Y 425.293,Z 441.133,A -85,B 0,C 180,E1 -9939.044,E2 -9939.044} C_VEL
LIN {X 0,Y 425.276,Z 441.137,A -85,B 0,C 180,E1 -9942.653,E2 -9942.653} C_VEL
LIN {X 0,Y 425.26,Z 441.14,A -85,B 0,C 180,E1 -9946.045,E2 -9946.045} C_VEL
LIN {X 0,Y 425.303,Z 441.132,A -85,B 0,C 180,E1 -9948.626,E2 -9948.626} C_VEL
LIN {X 0,Y 425.323,Z 441.13,A -85,B 0,C 180,E1 -9951.105,E2 -9951.105} C_VEL
LIN {X 0,Y 425.301,Z 441.132,A -85,B 0,C 180,E1 -9954.665,E2 -9954.665} C_VEL
LIN {X 0,Y 425.267,Z 441.139,A -85,B 0,C 180,E1 -9958.074,E2 -9958.074} C_VEL
LIN {X 0,Y 425.339,Z 441.129,A -85,B 0,C 180,E1 -9961.369,E2 -9961.369} C_VEL
LIN {X 0,Y 425.297,Z 441.133,A -85,B 0,C 180,E1 -9964.555,E2 -9964.555} C_VEL
LIN {X 0,Y 425.29,Z 441.137,A -85,B 0,C 180,E1 -9967.662,E2 -9967.662} C_VEL
LIN {X 0,Y 425.365,Z 441.124,A -85,B 0,C 180,E1 -9970.705,E2 -9970.705} C_VEL
LIN {X 0,Y 425.392,Z 441.123,A -85,B 0,C 180,E1 -9973.689,E2 -9973.689} C_VEL
LIN {X 0,Y 425.416,Z 441.121,A -85,B 0,C 180,E1 -9977.599,E2 -9977.599} C_VEL
LIN {X 0,Y 425.44,Z 441.119,A -85,B 0,C 180,E1 -9981.45,E2 -9981.45} C_VEL
LIN {X 0,Y 425.545,Z 441.102,A -85,B 0,C 180,E1 -9984.313,E2 -9984.313} C_VEL
LIN {X 0,Y 425.579,Z 441.098,A -85,B 0,C 180,E1 -9988.107,E2 -9988.107} C_VEL
LIN {X 0,Y 425.706,Z 441.081,A -85,B 0,C 180,E1 -9990,E2 -9990} C_VEL
LIN {X 0,Y 425.55,Z 441.103,A -85,B 0,C 180,E1 -9992.84,E2 -9992.84} C_VEL
LIN {X 0,Y 425.556,Z 441.102,A -85,B 0,C 180,E1 -9995.687,E2 -9995.687} C_VEL
LIN {X 0,Y 425.439,Z 441.115,A -85,B 0,C 180,E1 -9998.55,E2 -9998.55} C_VEL
LIN {X 0,Y 425.403,Z 441.119,A -85,B 0,C 180,E1 -9999.16,E2 -9999.16} C_VEL
LIN {X 0,Y 424.734,Z 441.205,A -85,B 0,C 180,E1 -9999.95,E2 -9999.95} C_VEL
LIN {X 0,Y 421.887,Z 441.561,A -85,B 0,C 180,E1 -10001.234,E2 -10001.234} C_VEL
LIN {X 0,Y 419.47,Z 441.861,A -85,B 0,C 180,E1 -10002.27,E2 -10002.27} C_VEL
LIN {X 0,Y 418.419,Z 441.992,A -85,B 0,C 180,E1 -10003.071,E2 -10003.071} C_VEL
LIN {X 0,Y 418.325,Z 442.002,A -85,B 0,C 180,E1 -10003.342,E2 -10003.342} C_VEL
LIN {X 0,Y 418.316,Z 442.004,A -85,B 0,C 180,E1 -10006.735,E2 -10006.735} C_VEL
LIN {X 0,Y 418.274,Z 442.008,A -85,B 0,C 180,E1 -10009.79,E2 -10009.79} C_VEL
LIN {X 0,Y 418.241,Z 442.013,A -85,B 0,C 180,E1 -10012.736,E2 -10012.736} C_VEL
LIN {X 0,Y 418.273,Z 442.007,A -85,B 0,C 180,E1 -10015.903,E2 -10015.903} C_VEL
LIN {X 0,Y 418.266,Z 442.01,A -85,B 0,C 180,E1 -10019.161,E2 -10019.161} C_VEL
LIN {X 0,Y 418.245,Z 442.015,A -85,B 0,C 180,E1 -10022.84,E2 -10022.84} C_VEL
LIN {X 0,Y 418.14,Z 442.028,A -85,B 0,C 180,E1 -10024.852,E2 -10024.852} C_VEL
LIN {X 0,Y 417.805,Z 442.067,A -85,B 0,C 180,E1 -10027.758,E2 -10027.758} C_VEL
LIN {X 0,Y 417.557,Z 442.102,A -85,B 0,C 180,E1 -10029.76,E2 -10029.76} C_VEL
LIN {X 0,Y 417.488,Z 442.702,A -85,B 0,C 180,E1 -10031.035,E2 -10031.035} C_VEL
LIN {X 0,Y 417.439,Z 445.027,A -85,B 0,C 180,E1 -10033.651,E2 -10033.651} C_VEL
LIN {X 0,Y 417.385,Z 447.508,A -85,B 0,C 180,E1 -10036.388,E2 -10036.388} C_VEL
LIN {X 0,Y 417.313,Z 450.157,A -85,B 0,C 180,E1 -10039.274,E2 -10039.274} C_VEL
LIN {X 0,Y 417.306,Z 452.125,A -85,B 0,C 180,E1 -10041.377,E2 -10041.377} C_VEL
LIN {X 0,Y 421.877,Z 468.585,A -85,B 0,C 180,E1 -10042.135,E2 -10042.135} C_VEL
LIN {X 0,Y 424.222,Z 478.061,A -85,B 0,C 180,E1 -10042.673,E2 -10042.673} C_VEL
LIN {X 0,Y 423.462,Z 492.178,A -85,B 0,C 180,E1 -10043.458,E2 -10043.458} C_VEL
LIN {X 0,Y 422.582,Z 505.36,A -85,B 0,C 180,E1 -10044.402,E2 -10044.402} C_VEL
LIN {X 0,Y 421.682,Z 517.446,A -85,B 0,C 180,E1 -10045.482,E2 -10045.482} C_VEL
LIN {X 0,Y 420.81,Z 527.961,A -85,B 0,C 180,E1 -10046.62,E2 -10046.62} C_VEL
LIN {X 0,Y 420.013,Z 538.069,A -85,B 0,C 180,E1 -10047.937,E2 -10047.937} C_VEL
LIN {X 0,Y 419.3,Z 546.561,A -85,B 0,C 180,E1 -10049.255,E2 -10049.255} C_VEL
LIN {X 0,Y 418.596,Z 555.158,A -85,B 0,C 180,E1 -10050.863,E2 -10050.863} C_VEL
LIN {X 0,Y 418.118,Z 562.159,A -85,B 0,C 180,E1 -10052.468,E2 -10052.468} C_VEL
LIN {X 0,Y 417.709,Z 567.805,A -85,B 0,C 180,E1 -10054.058,E2 -10054.058} C_VEL
LIN {X 0,Y 417.477,Z 571.553,A -85,B 0,C 180,E1 -10055.373,E2 -10055.373} C_VEL
LIN {X 0,Y 417.218,Z 575.617,A -85,B 0,C 180,E1 -10057.205,E2 -10057.205} C_VEL
LIN {X 0,Y 417.126,Z 577.342,A -85,B 0,C 180,E1 -10058.243,E2 -10058.243} C_VEL
LIN {X 0,Y 417.039,Z 578.664,A -85,B 0,C 180,E1 -10059.274,E2 -10059.274} C_VEL
LIN {X 0,Y 417.041,Z 579.788,A -85,B 0,C 180,E1 -10060.682,E2 -10060.682} C_VEL
LIN {X 0,Y 416.982,Z 580.247,A -85,B 0,C 180,E1 -10062.339,E2 -10062.339} C_VEL
LIN {X 0,Y 417.05,Z 579.448,A -85,B 0,C 180,E1 -10064.358,E2 -10064.358} C_VEL
LIN {X 0,Y 417.198,Z 577.215,A -85,B 0,C 180,E1 -10066.359,E2 -10066.359} C_VEL
LIN {X 0,Y 417.376,Z 575.136,A -85,B 0,C 180,E1 -10067.585,E2 -10067.585} C_VEL
LIN {X 0,Y 417.654,Z 571.107,A -85,B 0,C 180,E1 -10069.333,E2 -10069.333} C_VEL
LIN {X 0,Y 418.018,Z 566.657,A -85,B 0,C 180,E1 -10070.809,E2 -10070.809} C_VEL
LIN {X 0,Y 418.518,Z 560.349,A -85,B 0,C 180,E1 -10072.497,E2 -10072.497} C_VEL
LIN {X 0,Y 419.286,Z 552.296,A -85,B 0,C 180,E1 -10074.228,E2 -10074.228} C_VEL
LIN {X 0,Y 420.014,Z 544.029,A -85,B 0,C 180,E1 -10075.681,E2 -10075.681} C_VEL
LIN {X 0,Y 420.98,Z 534.05,A -85,B 0,C 180,E1 -10077.129,E2 -10077.129} C_VEL
LIN {X 0,Y 421.998,Z 522.825,A -85,B 0,C 180,E1 -10078.465,E2 -10078.465} C_VEL
LIN {X 0,Y 423.034,Z 510.719,A -85,B 0,C 180,E1 -10079.643,E2 -10079.643} C_VEL
LIN {X 0,Y 423.964,Z 498.69,A -85,B 0,C 180,E1 -10080.593,E2 -10080.593} C_VEL
LIN {X 0,Y 424.889,Z 485.282,A -85,B 0,C 180,E1 -10081.437,E2 -10081.437} C_VEL
LIN {X 0,Y 425.167,Z 479.43,A -85,B 0,C 180,E1 -10081.745,E2 -10081.745} C_VEL
LIN {X 0,Y 421.85,Z 467.225,A -85,B 0,C 180,E1 -10082.508,E2 -10082.508} C_VEL
LIN {X 0,Y 417.707,Z 455.268,A -85,B 0,C 180,E1 -10083.195,E2 -10083.195} C_VEL
LIN {X 0,Y 417.991,Z 454.02,A -85,B 0,C 180,E1 -10084.822,E2 -10084.822} C_VEL
LIN {X 0,Y 418.051,Z 451.917,A -85,B 0,C 180,E1 -10087.729,E2 -10087.729} C_VEL
LIN {X 0,Y 418.068,Z 449.912,A -85,B 0,C 180,E1 -10090.656,E2 -10090.656} C_VEL
LIN {X 0,Y 418.217,Z 448.432,A -85,B 0,C 180,E1 -10092.928,E2 -10092.928} C_VEL
LIN {X 0,Y 418.397,Z 446.103,A -85,B 0,C 180,E1 -10096.777,E2 -10096.777} C_VEL
LIN {X 0,Y 418.511,Z 444.444,A -85,B 0,C 180,E1 -10099.884,E2 -10099.884} C_VEL
LIN {X 0,Y 418.4,Z 443.206,A -85,B 0,C 180,E1 -10102.727,E2 -10102.727} C_VEL
LIN {X 0,Y 418.286,Z 442.134,A -85,B 0,C 180,E1 -10105.903,E2 -10105.903} C_VEL
LIN {X 0,Y 418.269,Z 442.011,A -85,B 0,C 180,E1 -10109.161,E2 -10109.161} C_VEL
LIN {X 0,Y 418.253,Z 442.012,A -85,B 0,C 180,E1 -10112.844,E2 -10112.844} C_VEL
LIN {X 0,Y 418.255,Z 442.012,A -85,B 0,C 180,E1 -10114.841,E2 -10114.841} C_VEL
LIN {X 0,Y 418.442,Z 443.01,A -85,B 0,C 180,E1 -10117.872,E2 -10117.872} C_VEL
LIN {X 0,Y 418.818,Z 444.933,A -85,B 0,C 180,E1 -10120.965,E2 -10120.965} C_VEL
LIN {X 0,Y 419.213,Z 447.472,A -85,B 0,C 180,E1 -10123.874,E2 -10123.874} C_VEL
LIN {X 0,Y 419.756,Z 450.542,A -85,B 0,C 180,E1 -10126.65,E2 -10126.65} C_VEL
LIN {X 0,Y 420.328,Z 454.063,A -85,B 0,C 180,E1 -10129.302,E2 -10129.302} C_VEL
LIN {X 0,Y 420.496,Z 457.894,A -85,B 0,C 180,E1 -10131.77,E2 -10131.77} C_VEL
LIN {X 0,Y 419.937,Z 462.123,A -85,B 0,C 180,E1 -10134.144,E2 -10134.144} C_VEL
LIN {X 0,Y 419.417,Z 467.439,A -85,B 0,C 180,E1 -10136.912,E2 -10136.912} C_VEL
LIN {X 0,Y 418.893,Z 474.568,A -85,B 0,C 180,E1 -10140.332,E2 -10140.332} C_VEL
LIN {X 0,Y 418.335,Z 481.78,A -85,B 0,C 180,E1 -10143.564,E2 -10143.564} C_VEL
LIN {X 0,Y 417.9,Z 490.436,A -85,B 0,C 180,E1 -10147.245,E2 -10147.245} C_VEL
LIN {X 0,Y 417.762,Z 494.162,A -85,B 0,C 180,E1 -10148.78,E2 -10148.78} C_VEL
LIN {X 0,Y 421.182,Z 510.164,A -85,B 0,C 180,E1 -10149.488,E2 -10149.488} C_VEL
LIN {X 0,Y 423.167,Z 524.852,A -85,B 0,C 180,E1 -10150.262,E2 -10150.262} C_VEL
LIN {X 0,Y 423.795,Z 530.966,A -85,B 0,C 180,E1 -10150.63,E2 -10150.63} C_VEL
LIN {X 0,Y 422.79,Z 544.658,A -85,B 0,C 180,E1 -10151.487,E2 -10151.487} C_VEL
LIN {X 0,Y 421.732,Z 558.026,A -85,B 0,C 180,E1 -10152.545,E2 -10152.545} C_VEL
LIN {X 0,Y 420.619,Z 570.328,A -85,B 0,C 180,E1 -10153.748,E2 -10153.748} C_VEL
LIN {X 0,Y 419.717,Z 580.569,A -85,B 0,C 180,E1 -10154.957,E2 -10154.957} C_VEL
LIN {X 0,Y 418.904,Z 590.84,A -85,B 0,C 180,E1 -10156.416,E2 -10156.416} C_VEL
LIN {X 0,Y 418.284,Z 599.443,A -85,B 0,C 180,E1 -10157.876,E2 -10157.876} C_VEL
LIN {X 0,Y 417.724,Z 607.698,A -85,B 0,C 180,E1 -10159.58,E2 -10159.58} C_VEL
LIN {X 0,Y 417.388,Z 614.376,A -85,B 0,C 180,E1 -10161.284,E2 -10161.284} C_VEL
LIN {X 0,Y 417.233,Z 620.323,A -85,B 0,C 180,E1 -10163.229,E2 -10163.229} C_VEL
LIN {X 0,Y 417.123,Z 624.658,A -85,B 0,C 180,E1 -10165.168,E2 -10165.168} C_VEL
LIN {X 0,Y 417.15,Z 627.512,A -85,B 0,C 180,E1 -10167.103,E2 -10167.103} C_VEL
LIN {X 0,Y 417.104,Z 628.93,A -85,B 0,C 180,E1 -10169.035,E2 -10169.035} C_VEL
LIN {X 0,Y 417.116,Z 628.947,A -85,B 0,C 180,E1 -10170.965,E2 -10170.965} C_VEL
LIN {X 0,Y 417.143,Z 627.571,A -85,B 0,C 180,E1 -10172.897,E2 -10172.897} C_VEL
LIN {X 0,Y 417.115,Z 624.769,A -85,B 0,C 180,E1 -10174.833,E2 -10174.833} C_VEL
LIN {X 0,Y 417.225,Z 620.474,A -85,B 0,C 180,E1 -10176.772,E2 -10176.772} C_VEL
LIN {X 0,Y 417.39,Z 614.557,A -85,B 0,C 180,E1 -10178.716,E2 -10178.716} C_VEL
LIN {X 0,Y 417.733,Z 607.879,A -85,B 0,C 180,E1 -10180.42,E2 -10180.42} C_VEL
LIN {X 0,Y 418.292,Z 599.567,A -85,B 0,C 180,E1 -10182.123,E2 -10182.123} C_VEL
LIN {X 0,Y 418.916,Z 590.881,A -85,B 0,C 180,E1 -10183.584,E2 -10183.584} C_VEL
LIN {X 0,Y 419.761,Z 580.379,A -85,B 0,C 180,E1 -10185.041,E2 -10185.041} C_VEL
LIN {X 0,Y 420.711,Z 568.683,A -85,B 0,C 180,E1 -10186.373,E2 -10186.373} C_VEL
LIN {X 0,Y 421.664,Z 557.059,A -85,B 0,C 180,E1 -10187.458,E2 -10187.458} C_VEL
LIN {X 0,Y 422.643,Z 544.377,A -85,B 0,C 180,E1 -10188.418,E2 -10188.418} C_VEL
LIN {X 0,Y 423.479,Z 530.098,A -85,B 0,C 180,E1 -10189.268,E2 -10189.268} C_VEL
LIN {X 0,Y 421.254,Z 515.303,A -85,B 0,C 180,E1 -10190.034,E2 -10190.034} C_VEL
LIN {X 0,Y 418.499,Z 500.814,A -85,B 0,C 180,E1 -10190.613,E2 -10190.613} C_VEL
LIN {X 0,Y 417.846,Z 496.992,A -85,B 0,C 180,E1 -10190.748,E2 -10190.748} C_VEL
LIN {X 0,Y 418.156,Z 489.703,A -85,B 0,C 180,E1 -10193.789,E2 -10193.789} C_VEL
LIN {X 0,Y 418.639,Z 481.77,A -85,B 0,C 180,E1 -10197.158,E2 -10197.158} C_VEL
LIN {X 0,Y 419.168,Z 473.641,A -85,B 0,C 180,E1 -10200.726,E2 -10200.726} C_VEL
LIN {X 0,Y 419.663,Z 467.372,A -85,B 0,C 180,E1 -10203.548,E2 -10203.548} C_VEL
LIN {X 0,Y 420.249,Z 459.964,A -85,B 0,C 180,E1 -10207.016,E2 -10207.016} C_VEL
LIN {X 0,Y 420.482,Z 456.238,A -85,B 0,C 180,E1 -10208.812,E2 -10208.812} C_VEL
LIN {X 0,Y 420.039,Z 451.684,A -85,B 0,C 180,E1 -10211.155,E2 -10211.155} C_VEL
LIN {X 0,Y 418.852,Z 445.008,A -85,B 0,C 180,E1 -10214.806,E2 -10214.806} C_VEL
LIN {X 0,Y 418.267,Z 442.008,A -85,B 0,C 180,E1 -10216.619,E2 -10216.619} C_VEL
LIN {X 0,Y 418.257,Z 442.011,A -85,B 0,C 180,E1 -10219.124,E2 -10219.124} C_VEL
LIN {X 0,Y 418.225,Z 442.017,A -85,B 0,C 180,E1 -10222.166,E2 -10222.166} C_VEL
LIN {X 0,Y 418.261,Z 442.011,A -85,B 0,C 180,E1 -10225.419,E2 -10225.419} C_VEL
LIN {X 0,Y 418.218,Z 442.015,A -85,B 0,C 180,E1 -10228.605,E2 -10228.605} C_VEL
LIN {X 0,Y 418.29,Z 442.005,A -85,B 0,C 180,E1 -10231.937,E2 -10231.937} C_VEL
LIN {X 0,Y 418.284,Z 442.009,A -85,B 0,C 180,E1 -10235.162,E2 -10235.162} C_VEL
LIN {X 0,Y 418.228,Z 442.014,A -85,B 0,C 180,E1 -10238.303,E2 -10238.303} C_VEL
LIN {X 0,Y 418.278,Z 442.007,A -85,B 0,C 180,E1 -10241.383,E2 -10241.383} C_VEL
LIN {X 0,Y 418.296,Z 442.007,A -85,B 0,C 180,E1 -10244.406,E2 -10244.406} C_VEL
LIN {X 0,Y 418.349,Z 441.999,A -85,B 0,C 180,E1 -10247.386,E2 -10247.386} C_VEL
LIN {X 0,Y 418.336,Z 442.001,A -85,B 0,C 180,E1 -10250.329,E2 -10250.329} C_VEL
LIN {X 0,Y 418.487,Z 441.982,A -85,B 0,C 180,E1 -10253.249,E2 -10253.249} C_VEL
LIN {X 0,Y 418.336,Z 442,A -85,B 0,C 180,E1 -10255.182,E2 -10255.182} C_VEL
LIN {X 0,Y 418.539,Z 441.976,A -85,B 0,C 180,E1 -10258.076,E2 -10258.076} C_VEL
LIN {X 0,Y 418.666,Z 441.958,A -85,B 0,C 180,E1 -10260,E2 -10260} C_VEL
LIN {X 0,Y 418.506,Z 441.981,A -85,B 0,C 180,E1 -10262.888,E2 -10262.888} C_VEL
LIN {X 0,Y 418.488,Z 441.982,A -85,B 0,C 180,E1 -10266.597,E2 -10266.597} C_VEL
LIN {X 0,Y 418.394,Z 441.995,A -85,B 0,C 180,E1 -10268.695,E2 -10268.695} C_VEL
LIN {X 0,Y 418.31,Z 442.003,A -85,B 0,C 180,E1 -10271.631,E2 -10271.631} C_VEL
LIN {X 0,Y 418.297,Z 442.007,A -85,B 0,C 180,E1 -10274.597,E2 -10274.597} C_VEL
LIN {X 0,Y 418.283,Z 442.006,A -85,B 0,C 180,E1 -10277.604,E2 -10277.604} C_VEL
LIN {X 0,Y 418.245,Z 442.014,A -85,B 0,C 180,E1 -10280.664,E2 -10280.664} C_VEL
LIN {X 0,Y 418.283,Z 442.008,A -85,B 0,C 180,E1 -10283.782,E2 -10283.782} C_VEL
LIN {X 0,Y 418.306,Z 442.002,A -85,B 0,C 180,E1 -10287.071,E2 -10287.071} C_VEL
LIN {X 0,Y 418.24,Z 442.015,A -85,B 0,C 180,E1 -10290.273,E2 -10290.273} C_VEL
LIN {X 0,Y 418.245,Z 442.013,A -85,B 0,C 180,E1 -10293.678,E2 -10293.678} C_VEL
LIN {X 0,Y 418.242,Z 442.011,A -85,B 0,C 180,E1 -10297.224,E2 -10297.224} C_VEL
LIN {X 0,Y 418.247,Z 442.012,A -85,B 0,C 180,E1 -10299.683,E2 -10299.683} C_VEL
LIN {X 0,Y 418.23,Z 442.015,A -85,B 0,C 180,E1 -10302.322,E2 -10302.322} C_VEL
LIN {X 0,Y 418.236,Z 442.011,A -85,B 0,C 180,E1 -10305.11,E2 -10305.11} C_VEL
LIN {X 0,Y 418.255,Z 442.012,A -85,B 0,C 180,E1 -10307.77,E2 -10307.77} C_VEL
LIN {X 0,Y 418.267,Z 442.009,A -85,B 0,C 180,E1 -10310.618,E2 -10310.618} C_VEL
LIN {X 0,Y 418.247,Z 442.014,A -85,B 0,C 180,E1 -10313.977,E2 -10313.977} C_VEL
LIN {X 0,Y 418.258,Z 442.01,A -85,B 0,C 180,E1 -10317.157,E2 -10317.157} C_VEL
LIN {X 0,Y 418.276,Z 442.007,A -85,B 0,C 180,E1 -10320.839,E2 -10320.839} C_VEL
LIN {X 0,Y 418.273,Z 442.009,A -85,B 0,C 180,E1 -10324.097,E2 -10324.097} C_VEL
LIN {X 0,Y 418.24,Z 442.012,A -85,B 0,C 180,E1 -10327.264,E2 -10327.264} C_VEL
LIN {X 0,Y 418.286,Z 442.006,A -85,B 0,C 180,E1 -10330.365,E2 -10330.365} C_VEL
LIN {X 0,Y 418.32,Z 442.005,A -85,B 0,C 180,E1 -10333.405,E2 -10333.405} C_VEL
LIN {X 0,Y 418.35,Z 441.998,A -85,B 0,C 180,E1 -10337,E2 -10337} C_VEL
LIN {X 0,Y 418.344,Z 441.998,A -85,B 0,C 180,E1 -10340.329,E2 -10340.329} C_VEL
LIN {X 0,Y 418.463,Z 441.987,A -85,B 0,C 180,E1 -10343.249,E2 -10343.249} C_VEL
LIN {X 0,Y 418.34,Z 442.001,A -85,B 0,C 180,E1 -10345.182,E2 -10345.182} C_VEL
LIN {X 0,Y 418.549,Z 441.974,A -85,B 0,C 180,E1 -10348.076,E2 -10348.076} C_VEL
LIN {X 0,Y 418.675,Z 441.957,A -85,B 0,C 180,E1 -10350,E2 -10350} C_VEL
LIN {X 0,Y 418.505,Z 441.981,A -85,B 0,C 180,E1 -10352.888,E2 -10352.888} C_VEL
LIN {X 0,Y 418.514,Z 441.979,A -85,B 0,C 180,E1 -10355.783,E2 -10355.783} C_VEL
LIN {X 0,Y 418.399,Z 441.992,A -85,B 0,C 180,E1 -10358.695,E2 -10358.695} C_VEL
LIN {X 0,Y 418.32,Z 442.004,A -85,B 0,C 180,E1 -10361.631,E2 -10361.631} C_VEL
LIN {X 0,Y 418.325,Z 442.002,A -85,B 0,C 180,E1 -10363.342,E2 -10363.342} C_VEL
LIN {X 0,Y 417.632,Z 442.088,A -85,B 0,C 180,E1 -10364.145,E2 -10364.145} C_VEL
LIN {X 0,Y 414.754,Z 442.448,A -85,B 0,C 180,E1 -10365.451,E2 -10365.451} C_VEL
LIN {X 0,Y 412.341,Z 442.747,A -85,B 0,C 180,E1 -10366.505,E2 -10366.505} C_VEL
LIN {X 0,Y 411.319,Z 442.877,A -85,B 0,C 180,E1 -10367.32,E2 -10367.32} C_VEL
LIN {X 0,Y 411.243,Z 442.881,A -85,B 0,C 180,E1 -10367.596,E2 -10367.596} C_VEL
LIN {X 0,Y 411.199,Z 442.891,A -85,B 0,C 180,E1 -10371.034,E2 -10371.034} C_VEL
LIN {X 0,Y 411.229,Z 442.885,A -85,B 0,C 180,E1 -10374.215,E2 -10374.215} C_VEL
LIN {X 0,Y 411.26,Z 442.882,A -85,B 0,C 180,E1 -10377.477,E2 -10377.477} C_VEL
LIN {X 0,Y 411.19,Z 442.892,A -85,B 0,C 180,E1 -10380.847,E2 -10380.847} C_VEL
LIN {X 0,Y 411.201,Z 442.89,A -85,B 0,C 180,E1 -10383.156,E2 -10383.156} C_VEL
LIN {X 0,Y 411.02,Z 442.913,A -85,B 0,C 180,E1 -10385.546,E2 -10385.546} C_VEL
LIN {X 0,Y 410.709,Z 442.951,A -85,B 0,C 180,E1 -10388.08,E2 -10388.08} C_VEL
LIN {X 0,Y 410.424,Z 443.046,A -85,B 0,C 180,E1 -10390.594,E2 -10390.594} C_VEL
LIN {X 0,Y 410.388,Z 445.366,A -85,B 0,C 180,E1 -10393.235,E2 -10393.235} C_VEL
LIN {X 0,Y 410.293,Z 448.508,A -85,B 0,C 180,E1 -10396.751,E2 -10396.751} C_VEL
LIN {X 0,Y 410.232,Z 450.928,A -85,B 0,C 180,E1 -10399.382,E2 -10399.382} C_VEL
LIN {X 0,Y 410.237,Z 452.605,A -85,B 0,C 180,E1 -10401.063,E2 -10401.063} C_VEL
LIN {X 0,Y 414.473,Z 467.728,A -85,B 0,C 180,E1 -10401.761,E2 -10401.761} C_VEL
LIN {X 0,Y 417.382,Z 479.073,A -85,B 0,C 180,E1 -10402.419,E2 -10402.419} C_VEL
LIN {X 0,Y 416.639,Z 492.952,A -85,B 0,C 180,E1 -10403.214,E2 -10403.214} C_VEL
LIN {X 0,Y 415.75,Z 505.8,A -85,B 0,C 180,E1 -10404.153,E2 -10404.153} C_VEL
LIN {X 0,Y 414.799,Z 518.052,A -85,B 0,C 180,E1 -10405.269,E2 -10405.269} C_VEL
LIN {X 0,Y 413.788,Z 529.768,A -85,B 0,C 180,E1 -10406.582,E2 -10406.582} C_VEL
LIN {X 0,Y 413.002,Z 539.335,A -85,B 0,C 180,E1 -10407.874,E2 -10407.874} C_VEL
LIN {X 0,Y 412.225,Z 547.843,A -85,B 0,C 180,E1 -10409.238,E2 -10409.238} C_VEL
LIN {X 0,Y 411.583,Z 555.751,A -85,B 0,C 180,E1 -10410.759,E2 -10410.759} C_VEL
LIN {X 0,Y 411.028,Z 563.148,A -85,B 0,C 180,E1 -10412.505,E2 -10412.505} C_VEL
LIN {X 0,Y 410.641,Z 568.681,A -85,B 0,C 180,E1 -10414.124,E2 -10414.124} C_VEL
LIN {X 0,Y 410.352,Z 573.053,A -85,B 0,C 180,E1 -10415.729,E2 -10415.729} C_VEL
LIN {X 0,Y 410.091,Z 577.017,A -85,B 0,C 180,E1 -10417.731,E2 -10417.731} C_VEL
LIN {X 0,Y 409.969,Z 578.644,A -85,B 0,C 180,E1 -10418.9,E2 -10418.9} C_VEL
LIN {X 0,Y 409.943,Z 580.372,A -85,B 0,C 180,E1 -10420.99,E2 -10420.99} C_VEL
LIN {X 0,Y 409.901,Z 580.599,A -85,B 0,C 180,E1 -10423.053,E2 -10423.053} C_VEL
LIN {X 0,Y 409.975,Z 580.144,A -85,B 0,C 180,E1 -10424.081,E2 -10424.081} C_VEL
LIN {X 0,Y 410.091,Z 578.141,A -85,B 0,C 180,E1 -10426.117,E2 -10426.117} C_VEL
LIN {X 0,Y 410.393,Z 574.674,A -85,B 0,C 180,E1 -10428.141,E2 -10428.141} C_VEL
LIN {X 0,Y 410.799,Z 569.693,A -85,B 0,C 180,E1 -10430.149,E2 -10430.149} C_VEL
LIN {X 0,Y 411.211,Z 564.857,A -85,B 0,C 180,E1 -10431.647,E2 -10431.647} C_VEL
LIN {X 0,Y 411.881,Z 557.895,A -85,B 0,C 180,E1 -10433.386,E2 -10433.386} C_VEL
LIN {X 0,Y 412.758,Z 549.294,A -85,B 0,C 180,E1 -10435.116,E2 -10435.116} C_VEL
LIN {X 0,Y 413.619,Z 540.34,A -85,B 0,C 180,E1 -10436.59,E2 -10436.59} C_VEL
LIN {X 0,Y 414.671,Z 529.502,A -85,B 0,C 180,E1 -10438.057,E2 -10438.057} C_VEL
LIN {X 0,Y 415.822,Z 517.353,A -85,B 0,C 180,E1 -10439.395,E2 -10439.395} C_VEL
LIN {X 0,Y 416.881,Z 505.216,A -85,B 0,C 180,E1 -10440.483,E2 -10440.483} C_VEL
LIN {X 0,Y 417.857,Z 492.122,A -85,B 0,C 180,E1 -10441.428,E2 -10441.428} C_VEL
LIN {X 0,Y 418.608,Z 481.342,A -85,B 0,C 180,E1 -10442.042,E2 -10442.042} C_VEL
LIN {X 0,Y 415.656,Z 470.132,A -85,B 0,C 180,E1 -10442.779,E2 -10442.779} C_VEL
LIN {X 0,Y 410.787,Z 456.117,A -85,B 0,C 180,E1 -10443.617,E2 -10443.617} C_VEL
LIN {X 0,Y 410.749,Z 455.817,A -85,B 0,C 180,E1 -10443.679,E2 -10443.679} C_VEL
LIN {X 0,Y 410.923,Z 454.195,A -85,B 0,C 180,E1 -10445.89,E2 -10445.89} C_VEL
LIN {X 0,Y 411.028,Z 452.127,A -85,B 0,C 180,E1 -10448.852,E2 -10448.852} C_VEL
LIN {X 0,Y 411.213,Z 449.542,A -85,B 0,C 180,E1 -10452.837,E2 -10452.837} C_VEL
LIN {X 0,Y 411.399,Z 447.15,A -85,B 0,C 180,E1 -10456.934,E2 -10456.934} C_VEL
LIN {X 0,Y 411.505,Z 445.579,A -85,B 0,C 180,E1 -10460.063,E2 -10460.063} C_VEL
LIN {X 0,Y 411.411,Z 444.324,A -85,B 0,C 180,E1 -10463.135,E2 -10463.135} C_VEL
LIN {X 0,Y 411.303,Z 443.38,A -85,B 0,C 180,E1 -10466.376,E2 -10466.376} C_VEL
LIN {X 0,Y 411.227,Z 442.895,A -85,B 0,C 180,E1 -10469.71,E2 -10469.71} C_VEL
LIN {X 0,Y 411.245,Z 443.051,A -85,B 0,C 180,E1 -10473.152,E2 -10473.152} C_VEL
LIN {X 0,Y 411.308,Z 443.623,A -85,B 0,C 180,E1 -10475.518,E2 -10475.518} C_VEL
LIN {X 0,Y 411.546,Z 444.748,A -85,B 0,C 180,E1 -10478.23,E2 -10478.23} C_VEL
LIN {X 0,Y 411.94,Z 446.785,A -85,B 0,C 180,E1 -10481.353,E2 -10481.353} C_VEL
LIN {X 0,Y 412.362,Z 449.447,A -85,B 0,C 180,E1 -10484.329,E2 -10484.329} C_VEL
LIN {X 0,Y 412.926,Z 452.549,A -85,B 0,C 180,E1 -10487.095,E2 -10487.095} C_VEL
LIN {X 0,Y 413.457,Z 456.328,A -85,B 0,C 180,E1 -10489.899,E2 -10489.899} C_VEL
LIN {X 0,Y 413.448,Z 460.063,A -85,B 0,C 180,E1 -10492.27,E2 -10492.27} C_VEL
LIN {X 0,Y 412.631,Z 466.439,A -85,B 0,C 180,E1 -10495.802,E2 -10495.802} C_VEL
LIN {X 0,Y 411.981,Z 473.23,A -85,B 0,C 180,E1 -10499.219,E2 -10499.219} C_VEL
LIN {X 0,Y 411.514,Z 479.118,A -85,B 0,C 180,E1 -10501.989,E2 -10501.989} C_VEL
LIN {X 0,Y 411.077,Z 485.8,A -85,B 0,C 180,E1 -10504.974,E2 -10504.974} C_VEL
LIN {X 0,Y 410.78,Z 493.811,A -85,B 0,C 180,E1 -10508.336,E2 -10508.336} C_VEL
LIN {X 0,Y 414.372,Z 510.066,A -85,B 0,C 180,E1 -10509.091,E2 -10509.091} C_VEL
LIN {X 0,Y 416.285,Z 524.195,A -85,B 0,C 180,E1 -10509.861,E2 -10509.861} C_VEL
LIN {X 0,Y 417.011,Z 532.346,A -85,B 0,C 180,E1 -10510.371,E2 -10510.371} C_VEL
LIN {X 0,Y 415.915,Z 546.03,A -85,B 0,C 180,E1 -10511.274,E2 -10511.274} C_VEL
LIN {X 0,Y 414.811,Z 559.21,A -85,B 0,C 180,E1 -10512.371,E2 -10512.371} C_VEL
LIN {X 0,Y 413.671,Z 571.193,A -85,B 0,C 180,E1 -10513.594,E2 -10513.594} C_VEL
LIN {X 0,Y 412.667,Z 582.128,A -85,B 0,C 180,E1 -10514.947,E2 -10514.947} C_VEL
LIN {X 0,Y 411.767,Z 592.68,A -85,B 0,C 180,E1 -10516.529,E2 -10516.529} C_VEL
LIN {X 0,Y 411.115,Z 601.637,A -85,B 0,C 180,E1 -10518.163,E2 -10518.163} C_VEL
LIN {X 0,Y 410.617,Z 608.373,A -85,B 0,C 180,E1 -10519.647,E2 -10519.647} C_VEL
LIN {X 0,Y 410.32,Z 613.995,A -85,B 0,C 180,E1 -10521.133,E2 -10521.133} C_VEL
LIN {X 0,Y 410.16,Z 619.94,A -85,B 0,C 180,E1 -10523.111,E2 -10523.111} C_VEL
LIN {X 0,Y 410.031,Z 624.269,A -85,B 0,C 180,E1 -10525.084,E2 -10525.084} C_VEL
LIN {X 0,Y 410.049,Z 627.109,A -85,B 0,C 180,E1 -10527.053,E2 -10527.053} C_VEL
LIN {X 0,Y 410.024,Z 628.511,A -85,B 0,C 180,E1 -10529.018,E2 -10529.018} C_VEL
LIN {X 0,Y 410.034,Z 628.515,A -85,B 0,C 180,E1 -10530.982,E2 -10530.982} C_VEL
LIN {X 0,Y 410.057,Z 627.124,A -85,B 0,C 180,E1 -10532.947,E2 -10532.947} C_VEL
LIN {X 0,Y 410.045,Z 624.305,A -85,B 0,C 180,E1 -10534.916,E2 -10534.916} C_VEL
LIN {X 0,Y 410.155,Z 619.987,A -85,B 0,C 180,E1 -10536.889,E2 -10536.889} C_VEL
LIN {X 0,Y 410.323,Z 614.04,A -85,B 0,C 180,E1 -10538.867,E2 -10538.867} C_VEL
LIN {X 0,Y 410.678,Z 607.326,A -85,B 0,C 180,E1 -10540.601,E2 -10540.601} C_VEL
LIN {X 0,Y 411.311,Z 598.955,A -85,B 0,C 180,E1 -10542.332,E2 -10542.332} C_VEL
LIN {X 0,Y 411.927,Z 590.211,A -85,B 0,C 180,E1 -10543.819,E2 -10543.819} C_VEL
